KUKA KRL program: MyProgram_082().src

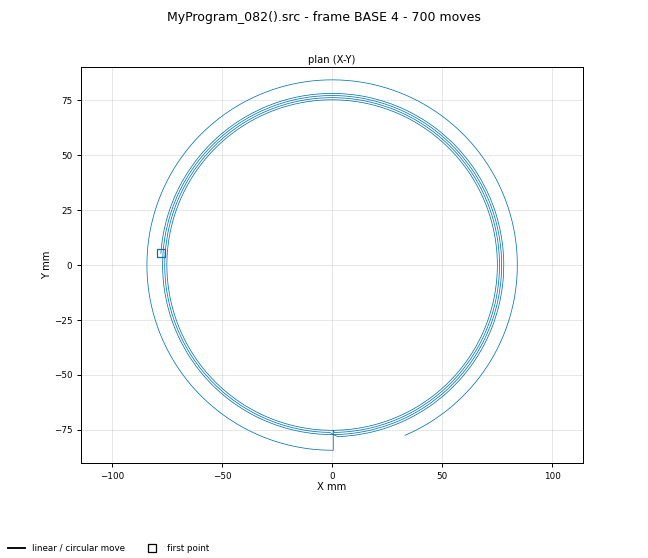
[picture p0: tool path of MyProgram_082().src in frame BASE 4, 700 of 700 moves have a stored position in this frame; points joined in program order, loops and branches not executed]
&ACCESS RVP
&REL 1
&PARAM TEMPLATE = C:\KRC\Roboter\Template\vorgabe
&PARAM EDITMASK = *
DEF MyProgram_082()
; ---- Setting reference (Base) ----
$BASE = BASE_DATA[4]

; --------------------------
; ---- Setting tool (TCP) ----
$TOOL = TOOL_DATA[3]
; --------------------------

$VEL.CP = VEL_APROX_PRINT
Startdeposition()
$VEL.CP = VEL_PRINT
LIN {X -77.8873,Y 5.2841,Z 82,A 170.2718,B 24.9035,C -2.2685,E1 24.8402,E2 274.3605} C_DIS
LIN {X -77.429,Y 9.9551,Z 82,A 166.7128,B 24.9028,C -2.2767,E1 24.8413,E2 277.9213} C_DIS
LIN {X -76.8059,Y 13.9726,Z 82,A 163.8687,B 24.9017,C -2.2896,E1 24.8426,E2 280.7516} C_DIS
LIN {X -76.3731,Y 16.1728,Z 82,A 161.8841,B 24.9019,C -2.2865,E1 24.8437,E2 282.7551} C_DIS
LIN {X -75.4009,Y 20.2256,Z 82,A 158.923,B 24.9009,C -2.2985,E1 24.8457,E2 285.7049} C_DIS
LIN {X -74.3801,Y 23.7078,Z 82,A 156.1268,B 24.9004,C -2.3035,E1 24.848,E2 288.5052} C_DIS
LIN {X -73.114,Y 27.3638,Z 82,A 153.5257,B 24.8992,C -2.318,E1 24.8504,E2 291.0865} C_DIS
LIN {X -71.5308,Y 31.2682,Z 82,A 150.0636,B 24.8992,C -2.3184,E1 24.8542,E2 294.567} C_DIS
LIN {X -69.857,Y 34.848,Z 82,A 147.6109,B 24.8975,C -2.3378,E1 24.8571,E2 296.9865} C_DIS
LIN {X -68.2862,Y 37.834,Z 82,A 144.7243,B 24.8977,C -2.335,E1 24.861,E2 299.8952} C_DIS
LIN {X -65.9152,Y 41.8294,Z 82,A 141.4118,B 24.8966,C -2.3469,E1 24.8657,E2 303.1961} C_DIS
LIN {X -62.1543,Y 47.2375,Z 82,A 136.7737,B 24.8951,C -2.3649,E1 24.8732,E2 307.8141} C_DIS
LIN {X -59.1537,Y 50.9447,Z 82,A 133.0603,B 24.8947,C -2.3686,E1 24.8798,E2 311.5357} C_DIS
LIN {X -56.492,Y 53.8793,Z 82,A 130.0106,B 24.8944,C -2.3723,E1 24.8856,E2 314.5901} C_DIS
LIN {X -53.6602,Y 56.7001,Z 82,A 126.9484,B 24.8941,C -2.376,E1 24.8917,E2 317.6562} C_DIS
LIN {X -50.9442,Y 59.1542,Z 82,A 124.7562,B 24.8924,C -2.3944,E1 24.8963,E2 319.8131} C_DIS
LIN {X -47.0479,Y 62.2967,Z 82,A 120.8026,B 24.8924,C -2.3952,E1 24.9049,E2 323.7796} C_DIS
LIN {X -43.5174,Y 64.8126,Z 82,A 117.5845,B 24.8919,C -2.4006,E1 24.9123,E2 326.9959} C_DIS
LIN {X -40.1757,Y 66.9348,Z 82,A 114.6066,B 24.8915,C -2.4041,E1 24.9194,E2 329.9747} C_DIS
LIN {X -36.2776,Y 69.1252,Z 82,A 111.3707,B 24.8909,C -2.4108,E1 24.9273,E2 333.2038} C_DIS
LIN {X -31.335,Y 71.5017,Z 82,A 107.627,B 24.8897,C -2.4243,E1 24.9367,E2 336.925} C_DIS
LIN {X -29.3343,Y 72.3454,Z 82,A 105.1652,B 24.8915,C -2.404,E1 24.9432,E2 339.4404} C_DIS
LIN {X -26.2143,Y 73.5344,Z 82,A 103.4691,B 24.8895,C -2.4267,E1 24.9475,E2 341.0861} C_DIS
LIN {X -23.2379,Y 74.5276,Z 82,A 100.9819,B 24.8897,C -2.4246,E1 24.9541,E2 343.5828} C_DIS
LIN {X -19.0837,Y 75.6986,Z 82,A 97.8114,B 24.8894,C -2.4277,E1 24.9627,E2 346.7507} C_DIS
LIN {X -15.9587,Y 76.4182,Z 82,A 94.8919,B 24.8906,C -2.4148,E1 24.9707,E2 349.7044} C_DIS
LIN {X -12.813,Y 77.0076,Z 82,A 92.4913,B 24.8906,C -2.4152,E1 24.9773,E2 352.1065} C_DIS
LIN {X -9.4491,Y 77.4932,Z 82,A 90.5626,B 24.889,C -2.4317,E1 24.9826,E2 353.9974} C_DIS
LIN {X -6.2457,Y 77.8161,Z 82,A 88.4719,B 24.8883,C -2.4401,E1 24.9883,E2 356.0689} C_DIS
LIN {X -2.6317,Y 78.0222,Z 82,A 85.4545,B 24.8891,C -2.4313,E1 24.9968,E2 359.1081} C_DIS
LIN {X 1.1853,Y 78.0577,Z 82,A 82.7985,B 24.8887,C -2.4358,E1 25.0042,E2 361.7533} C_DIS
LIN {X 4.2058,Y 77.953,Z 82,A 80.0123,B 24.8901,C -2.4204,E1 25.0121,E2 364.575} C_DIS
LIN {X 9.0381,Y 77.5414,Z 82,A 76.9843,B 24.8888,C -2.4345,E1 25.0204,E2 367.5677} C_DIS
LIN {X 12.3956,Y 77.0774,Z 82,A 74.4767,B 24.8888,C -2.4333,E1 25.0273,E2 370.0759} C_DIS
LIN {X 14.7919,Y 76.6521,Z 82,A 72.0569,B 24.8905,C -2.4151,E1 25.0341,E2 372.5362} C_DIS
LIN {X 18.2659,Y 75.8997,Z 82,A 69.8168,B 24.8897,C -2.4238,E1 25.0401,E2 374.7522} C_DIS
LIN {X 22.1454,Y 74.8594,Z 82,A 67.1483,B 24.8892,C -2.4297,E1 25.0472,E2 377.4025} C_DIS
LIN {X 27.0701,Y 73.2234,Z 82,A 63.363,B 24.8894,C -2.4271,E1 25.0572,E2 381.1863} C_DIS
LIN {X 30.8452,Y 71.7141,Z 82,A 60.3161,B 24.8899,C -2.4223,E1 25.0651,E2 384.2378} C_DIS
LIN {X 33.2005,Y 70.6552,Z 82,A 58.1622,B 24.8908,C -2.4127,E1 25.0706,E2 386.4089} C_DIS
LIN {X 36.1537,Y 69.1905,Z 82,A 55.6058,B 24.8914,C -2.4056,E1 25.0769,E2 388.9749} C_DIS
LIN {X 40.9292,Y 66.4769,Z 82,A 51.804,B 24.8914,C -2.4064,E1 25.086,E2 392.7631} C_DIS
LIN {X 43.8416,Y 64.5931,Z 82,A 49.597,B 24.8908,C -2.4122,E1 25.0911,E2 394.9491} C_DIS
LIN {X 46.4973,Y 62.7102,Z 82,A 47.0872,B 24.8915,C -2.4045,E1 25.0968,E2 397.4681} C_DIS
LIN {X 49.1805,Y 60.627,Z 82,A 44.682,B 24.8917,C -2.4026,E1 25.1021,E2 399.8689} C_DIS
LIN {X 53.8052,Y 56.5645,Z 82,A 40.1147,B 24.8926,C -2.3922,E1 25.1116,E2 404.4426} C_DIS
LIN {X 55.3996,Y 55.0025,Z 82,A 37.5288,B 24.8954,C -2.3608,E1 25.1168,E2 407.0916} C_DIS
LIN {X 58.5315,Y 51.6583,Z 82,A 35.1537,B 24.8935,C -2.3825,E1 25.1211,E2 409.405} C_DIS
LIN {X 62.0522,Y 47.3708,Z 82,A 31.4627,B 24.8933,C -2.3843,E1 25.1275,E2 413.0744} C_DIS
LIN {X 64.4349,Y 44.0753,Z 82,A 28.1614,B 24.8948,C -2.3674,E1 25.1329,E2 416.3998} C_DIS
LIN {X 66.1554,Y 41.4466,Z 82,A 25.946,B 24.8951,C -2.3642,E1 25.1362,E2 418.6115} C_DIS
LIN {X 67.7327,Y 38.8154,Z 82,A 23.6134,B 24.8959,C -2.3558,E1 25.1395,E2 420.952} C_DIS
LIN {X 70.3142,Y 33.9156,Z 82,A 20.0711,B 24.8954,C -2.3606,E1 25.1441,E2 424.4642} C_DIS
LIN {X 71.9062,Y 30.395,Z 82,A 16.8555,B 24.8972,C -2.341,E1 25.1478,E2 427.7087} C_DIS
LIN {X 72.9013,Y 27.9255,Z 82,A 14.8235,B 24.8979,C -2.3329,E1 25.1498,E2 429.7484} C_DIS
LIN {X 73.9869,Y 24.9056,Z 82,A 12.4921,B 24.8984,C -2.3267,E1 25.152,E2 432.0813} C_DIS
LIN {X 74.87,Y 22.1096,Z 82,A 9.9478,B 24.9,C -2.3083,E1 25.154,E2 434.6547} C_DIS
LIN {X 76.297,Y 16.5264,Z 82,A 5.6468,B 24.9013,C -2.2932,E1 25.1568,E2 438.9663} C_DIS
LIN {X 77.1156,Y 12.1461,Z 82,A 2.8117,B 24.9011,C -2.2965,E1 25.1581,E2 441.7772} C_DIS
LIN {X 77.5907,Y 8.6165,Z 82,A 0.0655,B 24.9021,C -2.2842,E1 25.1591,E2 444.5362} C_DIS
LIN {X 77.9848,Y 3.5743,Z 82,A -3.4052,B 24.9025,C -2.2799,E1 25.1597,E2 447.9965} C_DIS
LIN {X 78.0657,Y 0.3664,Z 82,A -5.5988,B 24.9027,C -2.2774,E1 25.1597,E2 450.1828} C_DIS
LIN {X 77.93,Y -4.6221,Z 82,A -9.3508,B 24.9039,C -2.2629,E1 25.1594,E2 453.9467} C_DIS
LIN {X 77.7316,Y -7.2215,Z 82,A -12.3122,B 24.9072,C -2.2246,E1 25.1586,E2 456.981} C_DIS
LIN {X 77.1522,Y -11.9113,Z 82,A -14.1609,B 24.9039,C -2.2635,E1 25.1579,E2 458.727} C_DIS
LIN {X 76.2149,Y -16.9028,Z 82,A -18.366,B 24.9061,C -2.2368,E1 25.1557,E2 462.9706} C_DIS
LIN {X 75.4606,Y -20.0044,Z 82,A -21.1675,B 24.9079,C -2.2153,E1 25.1537,E2 465.8068} C_DIS
LIN {X 73.6511,Y -25.8816,Z 82,A -25.0046,B 24.9074,C -2.2222,E1 25.1505,E2 469.6058} C_DIS
LIN {X 72.5926,Y -28.7174,Z 82,A -27.7071,B 24.9092,C -2.2005,E1 25.1477,E2 472.3443} C_DIS
LIN {X 70.4919,Y -33.5459,Z 82,A -31.2442,B 24.9092,C -2.199,E1 25.1437,E2 475.8658} C_DIS
LIN {X 68.5885,Y -37.2823,Z 82,A -34.6146,B 24.9108,C -2.1811,E1 25.1393,E2 479.2608} C_DIS
LIN {X 66.523,Y -40.8554,Z 82,A -37.3547,B 24.9108,C -2.1813,E1 25.1354,E2 481.9865} C_DIS
LIN {X 64.3814,Y -44.1542,Z 82,A -40.9192,B 24.9131,C -2.1526,E1 25.1297,E2 485.6009} C_DIS
LIN {X 62.2055,Y -47.1689,Z 82,A -43.079,B 24.9123,C -2.1626,E1 25.1262,E2 487.7269} C_DIS
LIN {X 60.5533,Y -49.2714,Z 82,A -45.6835,B 24.9143,C -2.138,E1 25.1215,E2 490.3773} C_DIS
LIN {X 57.8989,Y -52.3663,Z 82,A -47.3704,B 24.9117,C -2.17,E1 25.1185,E2 491.9812} C_DIS
LIN {X 54.1289,Y -56.2532,Z 82,A -51.2413,B 24.9122,C -2.1634,E1 25.111,E2 495.8511} C_DIS
LIN {X 51.7209,Y -58.4767,Z 82,A -54.1763,B 24.914,C -2.1417,E1 25.1049,E2 498.8254} C_DIS
LIN {X 50.0399,Y -59.9199,Z 82,A -56.6865,B 24.9164,C -2.1117,E1 25.0993,E2 501.3969} C_DIS
LIN {X 46.7247,Y -62.5396,Z 82,A -58.6933,B 24.9143,C -2.1378,E1 25.095,E2 503.3348} C_DIS
LIN {X 44.4197,Y -64.1966,Z 82,A -61.5923,B 24.9166,C -2.1093,E1 25.0883,E2 506.2912} C_DIS
LIN {X 41.5013,Y -66.1212,Z 82,A -63.0694,B 24.9144,C -2.1367,E1 25.085,E2 507.6985} C_DIS
LIN {X 39.5834,Y -67.2869,Z 82,A -65.7493,B 24.917,C -2.1031,E1 25.0783,E2 510.4498} C_DIS
LIN {X 36.6318,Y -68.9387,Z 82,A -67.7374,B 24.9162,C -2.1134,E1 25.0735,E2 512.4079} C_DIS
LIN {X 33.2308,Y -70.6411,Z 82,A -70.4044,B 24.9162,C -2.1126,E1 25.0668,E2 515.0698} C_DIS
LIN {X 30.2504,Y -71.9671,Z 82,A -72.9473,B 24.9169,C -2.1047,E1 25.0603,E2 517.6252} C_DIS
LIN {X 26.1878,Y -73.5436,Z 82,A -76.2474,B 24.9175,C -2.0975,E1 25.0516,E2 520.9354} C_DIS
LIN {X 23.3601,Y -74.4897,Z 82,A -78.4432,B 24.9177,C -2.0947,E1 25.0458,E2 523.1338} C_DIS
LIN {X 19.1921,Y -75.6708,Z 82,A -81.3872,B 24.9174,C -2.0981,E1 25.0379,E2 526.0649} C_DIS
LIN {X 15.9256,Y -76.425,Z 82,A -83.7655,B 24.9174,C -2.0983,E1 25.0314,E2 528.4398} C_DIS
LIN {X 9.9884,Y -77.4247,Z 82,A -87.7279,B 24.9167,C -2.1081,E1 25.0206,E2 532.3749} C_DIS
LIN {X 5.5408,Y -77.8699,Z 82,A -91.4789,B 24.9179,C -2.0929,E1 25.01,E2 536.1596} C_DIS
LIN {X 2.6008,Y -78.0232,Z 82,A -94.2473,B 24.9192,C -2.0752,E1 25.0022,E2 538.9694} C_DIS
LIN {X 2.6008,Y -78.0232,Z 82,A -94.2473,B 24.9192,C -2.0752,E1 25.0022,E2 538.9694} C_DIS
Enddeposition()
LIN {X 0.5081,Y -77.0915,Z 82,A -94.1358,B 24.9143,C -2.1379,E1 25.0029,E2 538.7091} C_DIS
Startdeposition()
$VEL.CP = VEL_PRINT
LIN {X 3.9501,Y -76.9968,Z 82,A -91.5866,B 24.9143,C -2.1385,E1 25.01,E2 536.1593} C_DIS
LIN {X 6.6748,Y -76.8091,Z 82,A -88.9999,B 24.9129,C -2.1554,E1 25.0173,E2 533.5338} C_DIS
LIN {X 10.5371,Y -76.3746,Z 82,A -86.2088,B 24.9129,C -2.1544,E1 25.0251,E2 530.7472} C_DIS
LIN {X 14.7289,Y -75.6776,Z 82,A -83.4663,B 24.9137,C -2.1449,E1 25.0325,E2 528.0303} C_DIS
LIN {X 17.832,Y -75.0082,Z 82,A -81.0789,B 24.9135,C -2.1479,E1 25.039,E2 525.6391} C_DIS
LIN {X 23.2313,Y -73.5153,Z 82,A -77.1971,B 24.9138,C -2.1443,E1 25.0494,E2 521.7725} C_DIS
LIN {X 28.0703,Y -71.8059,Z 82,A -73.1834,B 24.9129,C -2.1551,E1 25.06,E2 517.7415} C_DIS
LIN {X 30.9867,Y -70.5966,Z 82,A -70.8936,B 24.9128,C -2.1568,E1 25.0659,E2 515.4531} C_DIS
LIN {X 33.8173,Y -69.2864,Z 82,A -68.4579,B 24.9122,C -2.1639,E1 25.072,E2 513.0068} C_DIS
LIN {X 36.6293,Y -67.8405,Z 82,A -66.4322,B 24.9126,C -2.1583,E1 25.077,E2 511.0001} C_DIS
LIN {X 39.8423,Y -66.005,Z 82,A -63.7443,B 24.9124,C -2.1614,E1 25.0835,E2 508.313} C_DIS
LIN {X 42.2071,Y -64.5186,Z 82,A -61.3442,B 24.9113,C -2.175,E1 25.0892,E2 505.8885} C_DIS
LIN {X 44.9897,Y -62.61,Z 82,A -58.5122,B 24.91,C -2.1899,E1 25.0957,E2 503.0311} C_DIS
LIN {X 49.3722,Y -59.215,Z 82,A -54.9467,B 24.9107,C -2.182,E1 25.1034,E2 499.4976} C_DIS
LIN {X 51.4404,Y -57.4274,Z 82,A -52.997,B 24.9105,C -2.1841,E1 25.1075,E2 497.5506} C_DIS
LIN {X 53.2707,Y -55.7347,Z 82,A -50.8786,B 24.9095,C -2.1965,E1 25.1119,E2 495.4115} C_DIS
LIN {X 57.0794,Y -51.8277,Z 82,A -47.2458,B 24.9097,C -2.1936,E1 25.1189,E2 491.8013} C_DIS
LIN {X 60.3106,Y -48.0284,Z 82,A -42.4331,B 24.9061,C -2.2372,E1 25.1276,E2 486.9077} C_DIS
LIN {X 62.5808,Y -45.0302,Z 82,A -40.2831,B 24.9071,C -2.2248,E1 25.131,E2 484.7974} C_DIS
LIN {X 64.3492,Y -42.464,Z 82,A -37.5283,B 24.9055,C -2.2448,E1 25.1353,E2 482.009} C_DIS
LIN {X 66.0971,Y -39.6896,Z 82,A -35.7395,B 24.9066,C -2.2316,E1 25.1379,E2 480.2605} C_DIS
LIN {X 68.7522,Y -34.8884,Z 82,A -31.5814,B 24.9054,C -2.246,E1 25.1434,E2 476.0903} C_DIS
LIN {X 70.1743,Y -31.9321,Z 82,A -29.217,B 24.9049,C -2.2509,E1 25.1462,E2 473.7269} C_DIS
LIN {X 72.3496,Y -26.6385,Z 82,A -25.1385,B 24.9043,C -2.2584,E1 25.1504,E2 469.6533} C_DIS
LIN {X 73.4824,Y -23.335,Z 82,A -22.2849,B 24.9029,C -2.2744,E1 25.1529,E2 466.778} C_DIS
LIN {X 74.4554,Y -20.0105,Z 82,A -19.8348,B 24.9026,C -2.2786,E1 25.1548,E2 464.332} C_DIS
LIN {X 75.2068,Y -16.9735,Z 82,A -17.55,B 24.9021,C -2.2847,E1 25.1562,E2 462.0463} C_DIS
LIN {X 76.0528,Y -12.649,Z 82,A -14.4847,B 24.9017,C -2.2886,E1 25.1578,E2 458.9898} C_DIS
LIN {X 76.6432,Y -8.3636,Z 82,A -11.2642,B 24.9008,C -2.299,E1 25.159,E2 455.7637} C_DIS
LIN {X 76.8675,Y -5.953,Z 82,A -9.3343,B 24.9,C -2.3088,E1 25.1594,E2 453.8221} C_DIS
LIN {X 77.0423,Y -2.9386,Z 82,A -6.7313,B 24.8984,C -2.3271,E1 25.1597,E2 451.1911} C_DIS
LIN {X 77.0463,Y 2.8462,Z 82,A -3.0401,B 24.8989,C -2.3218,E1 25.1597,E2 447.5344} C_DIS
LIN {X 76.9112,Y 5.3576,Z 82,A -0.7479,B 24.8972,C -2.3409,E1 25.1592,E2 445.2108} C_DIS
LIN {X 76.5442,Y 9.2231,Z 82,A 2.5236,B 24.8953,C -2.362,E1 25.1582,E2 441.9087} C_DIS
LIN {X 76.0708,Y 12.541,Z 82,A 4.0458,B 24.8973,C -2.3397,E1 25.1576,E2 440.4483} C_DIS
LIN {X 75.6164,Y 15.0462,Z 82,A 7.107,B 24.8935,C -2.3818,E1 25.1559,E2 437.3054} C_DIS
LIN {X 74.7352,Y 18.9403,Z 82,A 8.8697,B 24.8961,C -2.3535,E1 25.1548,E2 435.6199} C_DIS
LIN {X 74.0877,Y 21.3339,Z 82,A 10.8114,B 24.8953,C -2.3621,E1 25.1533,E2 433.6691} C_DIS
LIN {X 73.3737,Y 23.6709,Z 82,A 12.8236,B 24.8943,C -2.3735,E1 25.1516,E2 431.6412} C_DIS
LIN {X 72.4155,Y 26.4578,Z 82,A 15.0029,B 24.8937,C -2.3796,E1 25.1495,E2 429.4598} C_DIS
LIN {X 71.3013,Y 29.3295,Z 82,A 17.6471,B 24.8922,C -2.3971,E1 25.1468,E2 426.7888} C_DIS
LIN {X 69.697,Y 32.9631,Z 82,A 20.2218,B 24.8925,C -2.3938,E1 25.1438,E2 424.236} C_DIS
LIN {X 67.8475,Y 36.6165,Z 82,A 22.9827,B 24.8925,C -2.3935,E1 25.1403,E2 421.4903} C_DIS
LIN {X 66.5797,Y 38.8758,Z 82,A 25.2155,B 24.8912,C -2.408,E1 25.1371,E2 419.235} C_DIS
LIN {X 64.7601,Y 41.8353,Z 82,A 27.5063,B 24.8914,C -2.4058,E1 25.1338,E2 416.9608} C_DIS
LIN {X 62.4871,Y 45.1598,Z 82,A 31.2112,B 24.8887,C -2.4349,E1 25.1277,E2 413.2053} C_DIS
LIN {X 59.1541,Y 49.4455,Z 82,A 34.5329,B 24.8898,C -2.4228,E1 25.122,E2 409.9276} C_DIS
LIN {X 57.415,Y 51.4542,Z 82,A 37.2241,B 24.8875,C -2.4488,E1 25.1169,E2 407.1869} C_DIS
LIN {X 53.7515,Y 55.2712,Z 82,A 40.6308,B 24.8881,C -2.4413,E1 25.1103,E2 403.8124} C_DIS
LIN {X 50.1748,Y 58.5368,Z 82,A 43.9057,B 24.8884,C -2.4388,E1 25.1035,E2 400.5565} C_DIS
LIN {X 48.2335,Y 60.1473,Z 82,A 46.0869,B 24.8872,C -2.4513,E1 25.0988,E2 398.354} C_DIS
LIN {X 45.8494,Y 61.9838,Z 82,A 48.3638,B 24.8867,C -2.4564,E1 25.0937,E2 396.0732} C_DIS
LIN {X 43.0679,Y 63.9469,Z 82,A 50.4983,B 24.8874,C -2.449,E1 25.0888,E2 393.9635} C_DIS
LIN {X 41.2641,Y 65.1268,Z 82,A 53.0326,B 24.8847,C -2.4788,E1 25.0827,E2 391.3669} C_DIS
LIN {X 38.4025,Y 66.8526,Z 82,A 55.4751,B 24.8845,C -2.4811,E1 25.0768,E2 388.9263} C_DIS
LIN {X 35.4552,Y 68.4625,Z 82,A 57.1028,B 24.8865,C -2.4591,E1 25.0729,E2 387.3552} C_DIS
LIN {X 33.035,Y 69.6625,Z 82,A 59.1236,B 24.8862,C -2.462,E1 25.0679,E2 385.3331} C_DIS
LIN {X 31.0756,Y 70.5578,Z 82,A 61.266,B 24.8846,C -2.4793,E1 25.0623,E2 383.1549} C_DIS
LIN {X 27.7636,Y 71.9264,Z 82,A 63.8133,B 24.8846,C -2.4786,E1 25.0557,E2 380.615} C_DIS
LIN {X 24.1282,Y 73.2258,Z 82,A 66.5464,B 24.8848,C -2.4771,E1 25.0485,E2 377.8906} C_DIS
LIN {X 19.882,Y 74.4901,Z 82,A 69.9019,B 24.8844,C -2.4812,E1 25.0395,E2 374.5312} C_DIS
LIN {X 15.6334,Y 75.4959,Z 82,A 72.5546,B 24.8858,C -2.4663,E1 25.0324,E2 371.9175} C_DIS
LIN {X 13.5841,Y 75.8913,Z 82,A 74.5578,B 24.8846,C -2.4795,E1 25.0268,E2 369.8852} C_DIS
LIN {X 10.6196,Y 76.3629,Z 82,A 76.7717,B 24.8846,C -2.4795,E1 25.0207,E2 367.6731} C_DIS
LIN {X 6.6725,Y 76.8088,Z 82,A 79.939,B 24.884,C -2.4859,E1 25.0118,E2 364.4928} C_DIS
LIN {X 3.8251,Y 77.0037,Z 82,A 81.9048,B 24.8844,C -2.4816,E1 25.0064,E2 362.5381} C_DIS
LIN {X 0.5366,Y 77.0956,Z 82,A 84.2089,B 24.8848,C -2.4774,E1 25,E2 360.2442} C_DIS
LIN {X -3.2844,Y 77.0275,Z 82,A 87.365,B 24.8841,C -2.4852,E1 24.9911,E2 357.0691} C_DIS
LIN {X -7.1127,Y 76.7687,Z 82,A 90.01,B 24.8847,C -2.4783,E1 24.9838,E2 354.4393} C_DIS
LIN {X -10.3824,Y 76.3966,Z 82,A 92.8584,B 24.8838,C -2.4877,E1 24.9758,E2 351.5666} C_DIS
LIN {X -15.1482,Y 75.5955,Z 82,A 95.7569,B 24.8858,C -2.4665,E1 24.968,E2 348.7156} C_DIS
LIN {X -17.6309,Y 75.055,Z 82,A 98.0189,B 24.8851,C -2.4747,E1 24.9618,E2 346.4311} C_DIS
LIN {X -20.9974,Y 74.183,Z 82,A 101.3824,B 24.8834,C -2.4928,E1 24.9526,E2 343.0193} C_DIS
LIN {X -24.8215,Y 72.9928,Z 82,A 103.2877,B 24.8863,C -2.4609,E1 24.9478,E2 341.1863} C_DIS
LIN {X -27.3843,Y 72.0702,Z 82,A 106.0937,B 24.8847,C -2.4788,E1 24.9403,E2 338.3318} C_DIS
LIN {X -32.2108,Y 70.0461,Z 82,A 109.7731,B 24.8857,C -2.4676,E1 24.9309,E2 334.6704} C_DIS
LIN {X -35.2561,Y 68.5643,Z 82,A 111.9235,B 24.887,C -2.4541,E1 24.9256,E2 332.5465} C_DIS
LIN {X -38.1112,Y 67.02,Z 82,A 114.8426,B 24.8861,C -2.463,E1 24.9185,E2 329.5977} C_DIS
LIN {X -41.7966,Y 64.7849,Z 82,A 117.5941,B 24.8878,C -2.4454,E1 24.912,E2 326.8793} C_DIS
LIN {X -44.3849,Y 63.0413,Z 82,A 120.0434,B 24.8878,C -2.4442,E1 24.9064,E2 324.4248} C_DIS
LIN {X -47.1418,Y 61.0055,Z 82,A 123.3863,B 24.8865,C -2.4592,E1 24.8989,E2 321.0337} C_DIS
LIN {X -50.3449,Y 58.3919,Z 82,A 125.3766,B 24.8896,C -2.4249,E1 24.8948,E2 319.1176} C_DIS
LIN {X -54.3022,Y 54.7295,Z 82,A 129.1584,B 24.891,C -2.41,E1 24.8871,E2 315.3559} C_DIS
LIN {X -57.8188,Y 51.0014,Z 82,A 133.4368,B 24.8908,C -2.4122,E1 24.8789,E2 311.0535} C_DIS
LIN {X -60.9616,Y 47.1988,Z 82,A 137.1674,B 24.8915,C -2.4043,E1 24.8724,E2 307.3244} C_DIS
LIN {X -63.7522,Y 43.3554,Z 82,A 140.5843,B 24.8926,C -2.392,E1 24.8669,E2 303.9202} C_DIS
LIN {X -65.29,Y 41.0033,Z 82,A 142.7697,B 24.8929,C -2.3885,E1 24.8636,E2 301.732} C_DIS
LIN {X -67.6657,Y 36.9516,Z 82,A 146.3026,B 24.8937,C -2.3796,E1 24.8587,E2 298.2021} C_DIS
LIN {X -69.1522,Y 34.0884,Z 82,A 148.7057,B 24.8944,C -2.3727,E1 24.8556,E2 295.8024} C_DIS
LIN {X -70.5534,Y 31.0858,Z 82,A 152.1596,B 24.8928,C -2.3899,E1 24.8517,E2 292.2886} C_DIS
LIN {X -72.1749,Y 27.108,Z 82,A 154.2774,B 24.8961,C -2.3537,E1 24.8496,E2 290.2454} C_DIS
LIN {X -73.3992,Y 23.5922,Z 82,A 157.5107,B 24.8958,C -2.3565,E1 24.8467,E2 286.9868} C_DIS
LIN {X -74.3415,Y 20.4323,Z 82,A 160.0168,B 24.8964,C -2.3503,E1 24.8448,E2 284.4811} C_DIS
LIN {X -75.5252,Y 15.4907,Z 82,A 163.3487,B 24.8984,C -2.3275,E1 24.8428,E2 281.1839} C_DIS
LIN {X -76.0455,Y 12.6924,Z 82,A 165.7516,B 24.8984,C -2.3278,E1 24.8416,E2 278.7661} C_DIS
LIN {X -76.5929,Y 8.8073,Z 82,A 168.7267,B 24.899,C -2.32,E1 24.8406,E2 275.7919} C_DIS
LIN {X -76.9455,Y 4.851,Z 82,A 171.6104,B 24.9,C -2.3089,E1 24.84,E2 272.9173} C_DIS
LIN {X -77.0936,Y 0.8846,Z 82,A 174.558,B 24.9008,C -2.2995,E1 24.8398,E2 269.9746} C_DIS
LIN {X -77.0556,Y -2.5454,Z 82,A 176.9796,B 24.9018,C -2.2883,E1 24.8399,E2 267.5651} C_DIS
LIN {X -76.8971,Y -5.5662,Z 82,A 179.4264,B 24.902,C -2.286,E1 24.8404,E2 265.1089} C_DIS
LIN {X -76.5566,Y -9.1173,Z 82,A -178.0985,B 24.903,C -2.2734,E1 24.8411,E2 262.6492} C_DIS
LIN {X -76.1375,Y -12.1339,Z 82,A -175.6368,B 24.9032,C -2.2712,E1 24.8421,E2 260.1781} C_DIS
LIN {X -75.4419,Y -15.8904,Z 82,A -172.8899,B 24.9042,C -2.2602,E1 24.8436,E2 257.4411} C_DIS
LIN {X -74.9446,Y -18.0929,Z 82,A -170.27,B 24.9026,C -2.2785,E1 24.8454,E2 254.7624} C_DIS
LIN {X -73.8516,Y -22.1361,Z 82,A -168.2018,B 24.9056,C -2.2432,E1 24.8469,E2 252.7664} C_DIS
LIN {X -73.0767,Y -24.5727,Z 82,A -166.0197,B 24.9055,C -2.2446,E1 24.8488,E2 250.5686} C_DIS
LIN {X -71.918,Y -27.7851,Z 82,A -162.5058,B 24.904,C -2.2616,E1 24.8524,E2 246.9941} C_DIS
LIN {X -70.1116,Y -32.0713,Z 82,A -160.0262,B 24.9069,C -2.2273,E1 24.8552,E2 244.5829} C_DIS
LIN {X -68.8561,Y -34.6851,Z 82,A -157.8851,B 24.9075,C -2.2211,E1 24.8578,E2 242.4452} C_DIS
LIN {X -65.8797,Y -40.0484,Z 82,A -153.5584,B 24.909,C -2.2031,E1 24.8638,E2 238.1386} C_DIS
LIN {X -64.4775,Y -42.2695,Z 82,A -150.3245,B 24.9067,C -2.2307,E1 24.8689,E2 234.8228} C_DIS
LIN {X -61.8304,Y -46.0556,Z 82,A -147.9294,B 24.9096,C -2.1958,E1 24.8727,E2 232.4994} C_DIS
LIN {X -59.8455,Y -48.606,Z 82,A -145.467,B 24.9099,C -2.1917,E1 24.877,E2 230.0352} C_DIS
LIN {X -57.9953,Y -50.7993,Z 82,A -142.8851,B 24.9093,C -2.1984,E1 24.8817,E2 227.4256} C_DIS
LIN {X -54.9121,Y -54.1173,Z 82,A -139.976,B 24.9109,C -2.1794,E1 24.8873,E2 224.5492} C_DIS
LIN {X -52.806,Y -56.1742,Z 82,A -137.2537,B 24.9101,C -2.1888,E1 24.8929,E2 221.7933} C_DIS
LIN {X -49.689,Y -58.9507,Z 82,A -134.6452,B 24.9117,C -2.17,E1 24.8983,E2 219.2194} C_DIS
LIN {X -47.1515,Y -60.9981,Z 82,A -131.6207,B 24.9107,C -2.1814,E1 24.9051,E2 216.1565} C_DIS
LIN {X -44.395,Y -63.0343,Z 82,A -129.1858,B 24.9113,C -2.1742,E1 24.9106,E2 213.7304} C_DIS
LIN {X -40.1524,Y -65.8165,Z 82,A -125.6154,B 24.9122,C -2.1633,E1 24.919,E2 210.1748} C_DIS
LIN {X -37.2718,Y -67.4905,Z 82,A -123.3806,B 24.913,C -2.1535,E1 24.9244,E2 207.9568} C_DIS
LIN {X -34.4211,Y -68.9873,Z 82,A -120.3806,B 24.9119,C -2.1668,E1 24.932,E2 204.9171} C_DIS
LIN {X -31.3077,Y -70.4555,Z 82,A -118.7273,B 24.9141,C -2.1396,E1 24.936,E2 203.3244} C_DIS
LIN {X -29.2523,Y -71.3327,Z 82,A -116.6037,B 24.9133,C -2.1504,E1 24.9416,E2 201.1703} C_DIS
LIN {X -25.4811,Y -72.7649,Z 82,A -113.5102,B 24.9133,C -2.1504,E1 24.9497,E2 198.0706} C_DIS
LIN {X -20.957,Y -74.1945,Z 82,A -109.8457,B 24.9132,C -2.1517,E1 24.9596,E2 194.3968} C_DIS
LIN {X -16.8908,Y -75.2258,Z 82,A -107.1236,B 24.9142,C -2.1392,E1 24.9669,E2 191.7008} C_DIS
LIN {X -13.867,Y -75.8404,Z 82,A -104.8342,B 24.9142,C -2.1383,E1 24.9732,E2 189.4111} C_DIS
LIN {X -9.6224,Y -76.4951,Z 82,A -101.3076,B 24.9136,C -2.1469,E1 24.983,E2 185.8612} C_DIS
LIN {X -5.6504,Y -76.8914,Z 82,A -98.6106,B 24.9142,C -2.1392,E1 24.9904,E2 183.1812} C_DIS
LIN {X -2.3423,Y -77.0619,Z 82,A -95.9455,B 24.9137,C -2.1452,E1 24.9979,E2 180.5014} C_DIS
LIN {X 0.5081,Y -77.0915,Z 82,A -94.1339,B 24.9143,C -2.1371,E1 25.0029,E2 178.7091} C_DIS
Enddeposition()
LIN {X 0.5081,Y -77.0915,Z 82,A -94.1339,B 24.9143,C -2.1371,E1 25.0029,E2 178.7091} C_DIS
Startdeposition()
$VEL.CP = VEL_PRINT
LIN {X -1.1038,Y -76.1212,Z 82,A -96.4432,B 24.9155,C -2.1232,E1 24.9964,E2 181.0513} C_DIS
LIN {X -4.2438,Y -76.0102,Z 82,A -98.8012,B 24.9155,C -2.1232,E1 24.9898,E2 183.4099} C_DIS
LIN {X -7.3852,Y -75.7705,Z 82,A -101.1105,B 24.9153,C -2.125,E1 24.9834,E2 185.7161} C_DIS
LIN {X -10.3028,Y -75.4293,Z 82,A -103.3603,B 24.9153,C -2.1243,E1 24.9771,E2 187.9691} C_DIS
LIN {X -12.9873,Y -75.0139,Z 82,A -105.4319,B 24.9153,C -2.1242,E1 24.9714,E2 190.043} C_DIS
LIN {X -15.9653,Y -74.4361,Z 82,A -107.7339,B 24.9153,C -2.1246,E1 24.9651,E2 192.3466} C_DIS
LIN {X -19.1563,Y -73.6793,Z 82,A -110.1969,B 24.9153,C -2.1261,E1 24.9584,E2 194.8095} C_DIS
LIN {X -22.2641,Y -72.8008,Z 82,A -113.4199,B 24.9167,C -2.1071,E1 24.9497,E2 198.083} C_DIS
LIN {X -25.8483,Y -71.6065,Z 82,A -115.7987,B 24.9156,C -2.1215,E1 24.9435,E2 200.4323} C_DIS
LIN {X -29.6391,Y -70.122,Z 82,A -118.6058,B 24.9148,C -2.1312,E1 24.9363,E2 203.2225} C_DIS
LIN {X -33.6955,Y -68.2656,Z 82,A -121.8468,B 24.9143,C -2.1381,E1 24.9281,E2 206.4554} C_DIS
LIN {X -36.3543,Y -66.8875,Z 82,A -123.9823,B 24.9138,C -2.144,E1 24.9229,E2 208.5827} C_DIS
LIN {X -40.4863,Y -64.4706,Z 82,A -127.7979,B 24.9138,C -2.1437,E1 24.9137,E2 212.4106} C_DIS
LIN {X -43.0643,Y -62.7791,Z 82,A -130.1727,B 24.9136,C -2.146,E1 24.9082,E2 214.7878} C_DIS
LIN {X -45.0341,Y -61.3799,Z 82,A -132.1209,B 24.9136,C -2.1459,E1 24.9038,E2 216.7433} C_DIS
LIN {X -47.941,Y -59.1373,Z 82,A -134.7189,B 24.9129,C -2.155,E1 24.8981,E2 219.3292} C_DIS
LIN {X -49.7768,Y -57.602,Z 82,A -137.2905,B 24.9142,C -2.1393,E1 24.8926,E2 221.9482} C_DIS
LIN {X -52.5194,Y -55.1131,Z 82,A -139.4131,B 24.9124,C -2.1613,E1 24.8883,E2 224.0272} C_DIS
LIN {X -54.8674,Y -52.7743,Z 82,A -141.4919,B 24.9111,C -2.1768,E1 24.8843,E2 226.0777} C_DIS
LIN {X -57.5803,Y -49.8016,Z 82,A -144.5728,B 24.9107,C -2.1822,E1 24.8785,E2 229.1595} C_DIS
LIN {X -59.9753,Y -46.8901,Z 82,A -147.616,B 24.9106,C -2.1838,E1 24.8732,E2 232.2131} C_DIS
LIN {X -62.2674,Y -43.8008,Z 82,A -150.7106,B 24.9104,C -2.186,E1 24.8681,E2 235.3175} C_DIS
LIN {X -64.0528,Y -41.1436,Z 82,A -152.946,B 24.9095,C -2.1963,E1 24.8646,E2 237.5395} C_DIS
LIN {X -65.5236,Y -38.7585,Z 82,A -155.0489,B 24.9091,C -2.2019,E1 24.8616,E2 239.6397} C_DIS
LIN {X -67.2626,Y -35.6559,Z 82,A -157.81,B 24.9086,C -2.2071,E1 24.8579,E2 242.4031} C_DIS
LIN {X -68.4668,Y -33.2864,Z 82,A -159.9208,B 24.9084,C -2.2099,E1 24.8553,E2 244.5184} C_DIS
LIN {X -70.1668,Y -29.5328,Z 82,A -163.0182,B 24.9077,C -2.2188,E1 24.8518,E2 247.6117} C_DIS
LIN {X -71.3749,Y -26.4832,Z 82,A -165.3887,B 24.9069,C -2.2282,E1 24.8494,E2 249.973} C_DIS
LIN {X -72.6497,Y -22.7515,Z 82,A -168.4579,B 24.9063,C -2.2346,E1 24.8467,E2 253.0445} C_DIS
LIN {X -73.5196,Y -19.7596,Z 82,A -171.2302,B 24.9066,C -2.2316,E1 24.8446,E2 255.8402} C_DIS
LIN {X -74.2607,Y -16.7645,Z 82,A -173.5501,B 24.906,C -2.2387,E1 24.8432,E2 258.1567} C_DIS
LIN {X -75.0464,Y -12.7931,Z 82,A -176.232,B 24.9045,C -2.2566,E1 24.8418,E2 260.8116} C_DIS
LIN {X -75.5002,Y -9.7612,Z 82,A -178.5431,B 24.9039,C -2.2638,E1 24.8409,E2 263.1195} C_DIS
LIN {X -75.8475,Y -6.5508,Z 82,A 178.8854,B 24.9035,C -2.2681,E1 24.8402,E2 265.6962} C_DIS
LIN {X -76.0581,Y -3.2761,Z 82,A 176.6134,B 24.9024,C -2.2805,E1 24.8399,E2 267.952} C_DIS
LIN {X -76.1275,Y -0.457,Z 82,A 174.3777,B 24.9021,C -2.2846,E1 24.8398,E2 270.1914} C_DIS
LIN {X -76.093,Y 2.3286,Z 82,A 172.2402,B 24.9016,C -2.2903,E1 24.8399,E2 272.3282} C_DIS
LIN {X -75.9285,Y 5.5293,Z 82,A 170.0202,B 24.9005,C -2.3025,E1 24.8403,E2 274.5324} C_DIS
LIN {X -75.7442,Y 7.6423,Z 82,A 167.6372,B 24.9017,C -2.2892,E1 24.841,E2 276.9614} C_DIS
LIN {X -74.8601,Y 13.8446,Z 82,A 163.6669,B 24.8989,C -2.3216,E1 24.8426,E2 280.8781} C_DIS
LIN {X -74.1373,Y 17.299,Z 82,A 160.2344,B 24.8997,C -2.3118,E1 24.8447,E2 284.3541} C_DIS
LIN {X -73.2757,Y 20.6457,Z 82,A 157.559,B 24.8992,C -2.3182,E1 24.8468,E2 287.0299} C_DIS
LIN {X -72.3265,Y 23.7605,Z 82,A 155.6664,B 24.8974,C -2.3387,E1 24.8483,E2 288.8842} C_DIS
LIN {X -71.2614,Y 26.7844,Z 82,A 153.2758,B 24.8967,C -2.3466,E1 24.8506,E2 291.2694} C_DIS
LIN {X -70.4557,Y 28.837,Z 82,A 151.3629,B 24.8967,C -2.3457,E1 24.8526,E2 293.1953} C_DIS
LIN {X -68.9697,Y 32.2298,Z 82,A 148.7727,B 24.8956,C -2.3586,E1 24.8556,E2 295.7687} C_DIS
LIN {X -67.6279,Y 34.9594,Z 82,A 146.5671,B 24.8948,C -2.3673,E1 24.8584,E2 297.9654} C_DIS
LIN {X -66.2025,Y 37.5891,Z 82,A 144.1623,B 24.8946,C -2.3701,E1 24.8616,E2 300.3761} C_DIS
LIN {X -64.5913,Y 40.2931,Z 82,A 141.8283,B 24.8939,C -2.3777,E1 24.865,E2 302.7041} C_DIS
LIN {X -62.8035,Y 43.0286,Z 82,A 139.2548,B 24.8936,C -2.3817,E1 24.869,E2 305.2808} C_DIS
LIN {X -59.9615,Y 46.9075,Z 82,A 135.6501,B 24.8927,C -2.3917,E1 24.875,E2 308.879} C_DIS
LIN {X -57.7965,Y 49.5497,Z 82,A 133.0908,B 24.892,C -2.3986,E1 24.8796,E2 311.4336} C_DIS
LIN {X -55.0325,Y 52.6026,Z 82,A 129.5255,B 24.8924,C -2.395,E1 24.8864,E2 315.0231} C_DIS
LIN {X -51.8034,Y 55.7869,Z 82,A 126.5102,B 24.8908,C -2.4126,E1 24.8925,E2 318.009} C_DIS
LIN {X -49.0785,Y 58.198,Z 82,A 123.6153,B 24.8906,C -2.4149,E1 24.8986,E2 320.9097} C_DIS
LIN {X -45.964,Y 60.6874,Z 82,A 120.8345,B 24.8895,C -2.4266,E1 24.9047,E2 323.6728} C_DIS
LIN {X -43.7567,Y 62.2981,Z 82,A 118.7603,B 24.8892,C -2.4303,E1 24.9094,E2 325.7454} C_DIS
LIN {X -41.1813,Y 64.0286,Z 82,A 116.4416,B 24.8887,C -2.4352,E1 24.9148,E2 328.0601} C_DIS
LIN {X -38.9491,Y 65.4109,Z 82,A 114.4534,B 24.8884,C -2.4384,E1 24.9195,E2 330.0466} C_DIS
LIN {X -36.3212,Y 66.9054,Z 82,A 112.2578,B 24.8879,C -2.4443,E1 24.9249,E2 332.2344} C_DIS
LIN {X -34.2684,Y 67.981,Z 82,A 110.4154,B 24.8879,C -2.4447,E1 24.9295,E2 334.081} C_DIS
LIN {X -31.5364,Y 69.29,Z 82,A 108.0973,B 24.8876,C -2.4472,E1 24.9353,E2 336.3989} C_DIS
LIN {X -27.1467,Y 71.1242,Z 82,A 104.5079,B 24.8872,C -2.4519,E1 24.9446,E2 339.9851} C_DIS
LIN {X -24.6322,Y 72.0342,Z 82,A 102.2196,B 24.8876,C -2.4474,E1 24.9507,E2 342.2886} C_DIS
LIN {X -20.3646,Y 73.3553,Z 82,A 99.3343,B 24.8861,C -2.4632,E1 24.9583,E2 345.1411} C_DIS
LIN {X -18.0173,Y 73.9658,Z 82,A 97.408,B 24.8861,C -2.4624,E1 24.9635,E2 347.072} C_DIS
LIN {X -14.9787,Y 74.6412,Z 82,A 94.7657,B 24.8867,C -2.4567,E1 24.9708,E2 349.7311} C_DIS
LIN {X -11.4059,Y 75.2696,Z 82,A 92.2099,B 24.8861,C -2.4632,E1 24.9778,E2 352.274} C_DIS
LIN {X -8.6608,Y 75.6346,Z 82,A 90.0277,B 24.8863,C -2.4618,E1 24.9839,E2 354.4609} C_DIS
LIN {X -5.3754,Y 75.9389,Z 82,A 87.6672,B 24.8858,C -2.4662,E1 24.9904,E2 356.8122} C_DIS
LIN {X -2.2406,Y 76.0957,Z 82,A 85.2457,B 24.8859,C -2.4654,E1 24.9972,E2 359.236} C_DIS
LIN {X 0.785,Y 76.1252,Z 82,A 82.9992,B 24.8859,C -2.4666,E1 25.0034,E2 361.4795} C_DIS
LIN {X 3.9006,Y 76.0292,Z 82,A 80.8215,B 24.8854,C -2.4712,E1 25.0095,E2 363.6455} C_DIS
LIN {X 5.9613,Y 75.8949,Z 82,A 79.1166,B 24.8858,C -2.4672,E1 25.0142,E2 365.3593} C_DIS
LIN {X 8.9002,Y 75.6065,Z 82,A 76.9406,B 24.8857,C -2.4681,E1 25.0203,E2 367.5316} C_DIS
LIN {X 12.0133,Y 75.1757,Z 82,A 74.6084,B 24.8857,C -2.4683,E1 25.0267,E2 369.8611} C_DIS
LIN {X 14.604,Y 74.715,Z 82,A 72.4547,B 24.8862,C -2.4629,E1 25.0327,E2 372.0253} C_DIS
LIN {X 17.6669,Y 74.0513,Z 82,A 70.0932,B 24.8862,C -2.4616,E1 25.0391,E2 374.3867} C_DIS
LIN {X 21.2159,Y 73.1131,Z 82,A 67.3566,B 24.8864,C -2.4605,E1 25.0464,E2 377.1214} C_DIS
LIN {X 25.9446,Y 71.5714,Z 82,A 63.707,B 24.8864,C -2.46,E1 25.0561,E2 380.7651} C_DIS
LIN {X 27.8209,Y 70.8629,Z 82,A 61.874,B 24.8874,C -2.4496,E1 25.0609,E2 382.6188} C_DIS
LIN {X 31.348,Y 69.3748,Z 82,A 59.2406,B 24.887,C -2.4533,E1 25.0676,E2 385.237} C_DIS
LIN {X 34.0422,Y 68.0937,Z 82,A 57.2872,B 24.8865,C -2.4587,E1 25.0725,E2 387.1723} C_DIS
LIN {X 37.5551,Y 66.222,Z 82,A 53.3617,B 24.8893,C -2.4286,E1 25.0822,E2 391.1577} C_DIS
LIN {X 40.5485,Y 64.4317,Z 82,A 51.5593,B 24.8875,C -2.4478,E1 25.0864,E2 392.9091} C_DIS
LIN {X 43.2075,Y 62.6798,Z 82,A 49.0319,B 24.8882,C -2.4402,E1 25.0923,E2 395.4459} C_DIS
LIN {X 45.8081,Y 60.8045,Z 82,A 46.6072,B 24.8887,C -2.4357,E1 25.0977,E2 397.8726} C_DIS
LIN {X 48.338,Y 58.8147,Z 82,A 44.1528,B 24.8892,C -2.4303,E1 25.1031,E2 400.3305} C_DIS
LIN {X 51.2875,Y 56.2602,Z 82,A 41.3115,B 24.8894,C -2.4273,E1 25.109,E2 403.1675} C_DIS
LIN {X 53.6936,Y 53.9688,Z 82,A 38.8551,B 24.8898,C -2.4234,E1 25.1139,E2 405.623} C_DIS
LIN {X 56.4711,Y 51.056,Z 82,A 35.7684,B 24.8905,C -2.4151,E1 25.1198,E2 408.7158} C_DIS
LIN {X 58.4795,Y 48.7413,Z 82,A 33.6377,B 24.8905,C -2.415,E1 25.1236,E2 410.8372} C_DIS
LIN {X 60.9698,Y 45.5881,Z 82,A 30.0376,B 24.8927,C -2.391,E1 25.1298,E2 414.4771} C_DIS
LIN {X 63.343,Y 42.2301,Z 82,A 27.3804,B 24.8923,C -2.396,E1 25.134,E2 417.1093} C_DIS
LIN {X 65.1981,Y 39.3044,Z 82,A 24.9163,B 24.8925,C -2.3934,E1 25.1376,E2 419.5669} C_DIS
LIN {X 66.6427,Y 36.8027,Z 82,A 22.8832,B 24.8926,C -2.3918,E1 25.1404,E2 421.5934} C_DIS
LIN {X 67.9044,Y 34.4182,Z 82,A 20.6736,B 24.8936,C -2.3809,E1 25.1433,E2 423.8169} C_DIS
LIN {X 69.0145,Y 32.1334,Z 82,A 18.3993,B 24.8951,C -2.3649,E1 25.146,E2 426.1169} C_DIS
LIN {X 70.7667,Y 28.0661,Z 82,A 15.4582,B 24.8949,C -2.367,E1 25.1491,E2 429.0368} C_DIS
LIN {X 71.8655,Y 25.1182,Z 82,A 13.2078,B 24.8952,C -2.3636,E1 25.1513,E2 431.2827} C_DIS
LIN {X 72.7828,Y 22.3221,Z 82,A 10.8003,B 24.8963,C -2.3512,E1 25.1533,E2 433.7057} C_DIS
LIN {X 73.6595,Y 19.2334,Z 82,A 8.829,B 24.8957,C -2.3573,E1 25.1548,E2 435.6513} C_DIS
LIN {X 74.3247,Y 16.4762,Z 82,A 6.3709,B 24.8972,C -2.341,E1 25.1563,E2 438.1336} C_DIS
LIN {X 74.9946,Y 13.0966,Z 82,A 3.7878,B 24.8978,C -2.3333,E1 25.1577,E2 440.7198} C_DIS
LIN {X 75.4727,Y 9.9737,Z 82,A 1.1791,B 24.8991,C -2.319,E1 25.1587,E2 443.347} C_DIS
LIN {X 75.8876,Y 6.0525,Z 82,A -1.3986,B 24.8989,C -2.3214,E1 25.1594,E2 445.9037} C_DIS
LIN {X 76.0663,Y 3.085,Z 82,A -3.5635,B 24.8993,C -2.3165,E1 25.1597,E2 448.0674} C_DIS
LIN {X 76.1285,Y 0.2682,Z 82,A -5.8556,B 24.9004,C -2.3045,E1 25.1597,E2 450.374} C_DIS
LIN {X 76.0728,Y -2.9326,Z 82,A -8.2489,B 24.901,C -2.2973,E1 25.1596,E2 452.7701} C_DIS
LIN {X 75.9009,Y -5.8855,Z 82,A -10.3757,B 24.9013,C -2.2932,E1 25.1592,E2 454.894} C_DIS
LIN {X 75.6397,Y -8.617,Z 82,A -12.2727,B 24.9015,C -2.2917,E1 25.1587,E2 456.7833} C_DIS
LIN {X 75.2823,Y -11.3238,Z 82,A -14.545,B 24.9026,C -2.2786,E1 25.1578,E2 459.0731} C_DIS
LIN {X 74.6728,Y -14.8229,Z 82,A -17.2505,B 24.9034,C -2.2692,E1 25.1564,E2 461.7852} C_DIS
LIN {X 74.073,Y -17.5771,Z 82,A -19.3063,B 24.9038,C -2.2644,E1 25.1551,E2 463.8401} C_DIS
LIN {X 73.3717,Y -20.3059,Z 82,A -21.4496,B 24.9044,C -2.2571,E1 25.1536,E2 465.9885} C_DIS
LIN {X 72.5994,Y -22.9137,Z 82,A -23.2282,B 24.9043,C -2.2589,E1 25.1521,E2 467.7528} C_DIS
LIN {X 71.6825,Y -25.6395,Z 82,A -25.369,B 24.9048,C -2.2529,E1 25.1502,E2 469.8957} C_DIS
LIN {X 70.3947,Y -28.9869,Z 82,A -28.137,B 24.9057,C -2.2426,E1 25.1474,E2 472.6726} C_DIS
LIN {X 69.2061,Y -31.7216,Z 82,A -30.4753,B 24.9065,C -2.233,E1 25.1447,E2 475.0208} C_DIS
LIN {X 67.9283,Y -34.3716,Z 82,A -32.3676,B 24.9062,C -2.2362,E1 25.1424,E2 476.8955} C_DIS
LIN {X 66.7538,Y -36.6,Z 82,A -34.4996,B 24.9073,C -2.2235,E1 25.1395,E2 479.0461} C_DIS
LIN {X 65.517,Y -38.7696,Z 82,A -36.6244,B 24.9083,C -2.2108,E1 25.1365,E2 481.1901} C_DIS
LIN {X 62.9771,Y -42.7722,Z 82,A -40.41,B 24.9097,C -2.1944,E1 25.1307,E2 484.9955} C_DIS
LIN {X 59.6418,Y -47.3121,Z 82,A -44.2284,B 24.9096,C -2.1956,E1 25.1243,E2 488.7929} C_DIS
LIN {X 57.6145,Y -49.7625,Z 82,A -46.6947,B 24.9103,C -2.1872,E1 25.1198,E2 491.2677} C_DIS
LIN {X 54.97,Y -52.668,Z 82,A -49.5045,B 24.9105,C -2.1843,E1 25.1145,E2 494.0722} C_DIS
LIN {X 52.7765,Y -54.8653,Z 82,A -51.8549,B 24.911,C -2.1783,E1 25.1098,E2 496.4269} C_DIS
LIN {X 50.399,Y -57.0586,Z 82,A -54.3454,B 24.9116,C -2.171,E1 25.1046,E2 498.9246} C_DIS
LIN {X 47.4528,Y -59.5306,Z 82,A -57.4936,B 24.9127,C -2.1573,E1 25.0978,E2 502.0933} C_DIS
LIN {X 44.2286,Y -61.9628,Z 82,A -60.3539,B 24.9127,C -2.1562,E1 25.0914,E2 504.9461} C_DIS
LIN {X 40.2314,Y -64.6298,Z 82,A -63.1553,B 24.9114,C -2.1729,E1 25.085,E2 507.6985} C_DIS
LIN {X 37.488,Y -66.2597,Z 82,A -66.2285,B 24.9134,C -2.149,E1 25.0774,E2 510.8189} C_DIS
LIN {X 34.673,Y -67.7742,Z 82,A -68.4677,B 24.9134,C -2.1498,E1 25.0719,E2 513.0501} C_DIS
LIN {X 32.2074,Y -68.9801,Z 82,A -70.5452,B 24.9136,C -2.1462,E1 25.0667,E2 515.1307} C_DIS
LIN {X 29.663,Y -70.1119,Z 82,A -72.7046,B 24.914,C -2.1413,E1 25.0611,E2 517.2965} C_DIS
LIN {X 26.943,Y -71.2014,Z 82,A -74.6893,B 24.9137,C -2.1445,E1 25.056,E2 519.2691} C_DIS
LIN {X 23.7034,Y -72.3449,Z 82,A -77.1506,B 24.9137,C -2.1448,E1 25.0495,E2 521.7249} C_DIS
LIN {X 20.9964,Y -73.1763,Z 82,A -79.569,B 24.9146,C -2.1342,E1 25.043,E2 524.164} C_DIS
LIN {X 18.3121,Y -73.8939,Z 82,A -81.7282,B 24.9149,C -2.1302,E1 25.0371,E2 526.3294} C_DIS
LIN {X 15.4942,Y -74.5354,Z 82,A -83.8318,B 24.9149,C -2.1302,E1 25.0314,E2 528.4303} C_DIS
LIN {X 12.6272,Y -75.0741,Z 82,A -86.0444,B 24.9151,C -2.128,E1 25.0253,E2 530.6457} C_DIS
LIN {X 9.8976,Y -75.4825,Z 82,A -88.257,B 24.9155,C -2.1229,E1 25.0192,E2 532.8685} C_DIS
LIN {X 6.4315,Y -75.8573,Z 82,A -90.8101,B 24.9155,C -2.1234,E1 25.0121,E2 535.4188} C_DIS
LIN {X 3.3236,Y -76.056,Z 82,A -92.9818,B 24.9151,C -2.1272,E1 25.0061,E2 537.5806} C_DIS
LIN {X 0.9531,Y -76.1239,Z 82,A -95.0936,B 24.9159,C -2.1178,E1 25.0001,E2 539.7146} C_DIS
LIN {X 0.9531,Y -76.1239,Z 82,A -95.0936,B 24.9159,C -2.1178,E1 25.0001,E2 539.7146} C_DIS
Enddeposition()
LIN {X 0.5084,Y -75.156,Z 82,A -95.0256,B 24.9137,C -2.1457,E1 25.0005,E2 539.5804} C_DIS
Startdeposition()
$VEL.CP = VEL_PRINT
LIN {X 2.4777,Y -75.1191,Z 82,A -92.6783,B 24.9117,C -2.1692,E1 25.0072,E2 537.1777} C_DIS
LIN {X 5.5231,Y -74.9579,Z 82,A -90.2948,B 24.9115,C -2.1718,E1 25.0138,E2 534.7891} C_DIS
LIN {X 8.5586,Y -74.6711,Z 82,A -88.0525,B 24.9116,C -2.1708,E1 25.0201,E2 532.5505} C_DIS
LIN {X 11.6462,Y -74.2521,Z 82,A -85.8136,B 24.9118,C -2.1686,E1 25.0262,E2 530.3188} C_DIS
LIN {X 14.3785,Y -73.7718,Z 82,A -83.7076,B 24.9117,C -2.1701,E1 25.032,E2 528.2117} C_DIS
LIN {X 17.0779,Y -73.194,Z 82,A -81.6063,B 24.9115,C -2.1719,E1 25.0377,E2 526.1089} C_DIS
LIN {X 19.7539,Y -72.5175,Z 82,A -79.5058,B 24.9114,C -2.174,E1 25.0434,E2 524.0067} C_DIS
LIN {X 22.0758,Y -71.8448,Z 82,A -77.5259,B 24.9109,C -2.1799,E1 25.0487,E2 522.0161} C_DIS
LIN {X 25.064,Y -70.8577,Z 82,A -75.2726,B 24.9109,C -2.1788,E1 25.0547,E2 519.77} C_DIS
LIN {X 27.3293,Y -70.0151,Z 82,A -73.3062,B 24.9105,C -2.1848,E1 25.0598,E2 517.7936} C_DIS
LIN {X 29.881,Y -68.9647,Z 82,A -71.2101,B 24.9102,C -2.1876,E1 25.0652,E2 515.6957} C_DIS
LIN {X 32.7006,Y -67.6733,Z 82,A -68.9851,B 24.9102,C -2.1873,E1 25.0708,E2 513.4772} C_DIS
LIN {X 35.1625,Y -66.4275,Z 82,A -66.7377,B 24.9096,C -2.195,E1 25.0765,E2 511.2179} C_DIS
LIN {X 37.8266,Y -64.9486,Z 82,A -64.3549,B 24.9091,C -2.2008,E1 25.0822,E2 508.8283} C_DIS
LIN {X 40.2045,Y -63.5042,Z 82,A -62.2515,B 24.9089,C -2.2043,E1 25.0872,E2 506.7235} C_DIS
LIN {X 42.4911,Y -61.9973,Z 82,A -60.2997,B 24.9089,C -2.2044,E1 25.0917,E2 504.7778} C_DIS
LIN {X 44.7113,Y -60.4155,Z 82,A -58.0808,B 24.9081,C -2.2129,E1 25.0968,E2 502.5469} C_DIS
LIN {X 47.2827,Y -58.4237,Z 82,A -55.6864,B 24.9079,C -2.2157,E1 25.102,E2 500.1547} C_DIS
LIN {X 49.6865,Y -56.3945,Z 82,A -53.2738,B 24.9074,C -2.2215,E1 25.1071,E2 497.7378} C_DIS
LIN {X 51.9312,Y -54.3345,Z 82,A -50.9778,B 24.907,C -2.2262,E1 25.1118,E2 495.4402} C_DIS
LIN {X 54.0085,Y -52.2694,Z 82,A -48.8361,B 24.9068,C -2.2289,E1 25.116,E2 493.3012} C_DIS
LIN {X 55.9977,Y -50.1322,Z 82,A -46.5705,B 24.9062,C -2.2357,E1 25.1203,E2 491.0296} C_DIS
LIN {X 58.0101,Y -47.7903,Z 82,A -44.2428,B 24.9058,C -2.241,E1 25.1245,E2 488.7001} C_DIS
LIN {X 59.8453,Y -45.4719,Z 82,A -41.9377,B 24.9052,C -2.2485,E1 25.1284,E2 486.3881} C_DIS
LIN {X 61.4589,Y -43.2664,Z 82,A -39.8565,B 24.9047,C -2.2541,E1 25.1318,E2 484.3038} C_DIS
LIN {X 62.9935,Y -41,Z 82,A -37.7812,B 24.9042,C -2.2595,E1 25.135,E2 482.2259} C_DIS
LIN {X 64.4421,Y -38.683,Z 82,A -35.7191,B 24.9038,C -2.2648,E1 25.138,E2 480.1618} C_DIS
LIN {X 65.924,Y -36.0985,Z 82,A -33.4736,B 24.9033,C -2.2706,E1 25.1411,E2 477.9143} C_DIS
LIN {X 67.4161,Y -33.2276,Z 82,A -31.2149,B 24.9032,C -2.2716,E1 25.1439,E2 475.6653} C_DIS
LIN {X 68.5903,Y -30.7308,Z 82,A -29.124,B 24.9027,C -2.2775,E1 25.1464,E2 473.5718} C_DIS
LIN {X 69.6717,Y -28.1933,Z 82,A -27.0339,B 24.9022,C -2.2835,E1 25.1486,E2 471.4791} C_DIS
LIN {X 70.6682,Y -25.5934,Z 82,A -24.9282,B 24.9017,C -2.2894,E1 25.1507,E2 469.371} C_DIS
LIN {X 71.5671,Y -22.96,Z 82,A -22.6637,B 24.9007,C -2.3003,E1 25.1527,E2 467.0936} C_DIS
LIN {X 72.4404,Y -20.0396,Z 82,A -20.2991,B 24.9,C -2.3088,E1 25.1545,E2 464.7224} C_DIS
LIN {X 73.1273,Y -17.3665,Z 82,A -18.2076,B 24.8994,C -2.3151,E1 25.1559,E2 462.6283} C_DIS
LIN {X 73.7155,Y -14.6699,Z 82,A -16.1196,B 24.8989,C -2.3212,E1 25.1571,E2 460.5379} C_DIS
LIN {X 74.251,Y -11.6534,Z 82,A -13.8746,B 24.8985,C -2.3259,E1 25.1581,E2 458.2951} C_DIS
LIN {X 74.6703,Y -8.5647,Z 82,A -11.6553,B 24.8982,C -2.3287,E1 25.1589,E2 456.0822} C_DIS
LIN {X 74.9344,Y -5.818,Z 82,A -9.5679,B 24.8977,C -2.3349,E1 25.1594,E2 453.9925} C_DIS
LIN {X 75.0828,Y -3.4049,Z 82,A -7.6019,B 24.8969,C -2.3445,E1 25.1597,E2 452.0154} C_DIS
LIN {X 75.1587,Y -0.4421,Z 82,A -5.4338,B 24.8965,C -2.349,E1 25.1597,E2 449.8498} C_DIS
LIN {X 75.119,Y 2.4807,Z 82,A -3.1259,B 24.8956,C -2.3585,E1 25.1597,E2 447.5333} C_DIS
LIN {X 74.958,Y 5.5218,Z 82,A -0.7605,B 24.8949,C -2.3671,E1 25.1592,E2 445.1614} C_DIS
LIN {X 74.6718,Y 8.5525,Z 82,A 1.4673,B 24.8945,C -2.3716,E1 25.1586,E2 442.9362} C_DIS
LIN {X 74.2503,Y 11.6582,Z 82,A 3.7011,B 24.8942,C -2.3744,E1 25.1577,E2 440.7091} C_DIS
LIN {X 73.7726,Y 14.3738,Z 82,A 5.7898,B 24.8937,C -2.3805,E1 25.1566,E2 438.6182} C_DIS
LIN {X 73.1959,Y 17.0697,Z 82,A 7.8788,B 24.8931,C -2.3865,E1 25.1554,E2 436.527} C_DIS
LIN {X 72.5149,Y 19.7636,Z 82,A 9.9845,B 24.8926,C -2.3926,E1 25.1539,E2 434.4191} C_DIS
LIN {X 71.8383,Y 22.0968,Z 82,A 11.9537,B 24.8918,C -2.4016,E1 25.1523,E2 432.4398} C_DIS
LIN {X 70.8644,Y 25.0449,Z 82,A 14.1727,B 24.8915,C -2.4042,E1 25.1503,E2 430.2273} C_DIS
LIN {X 70.0212,Y 27.3139,Z 82,A 16.1249,B 24.8908,C -2.4127,E1 25.1483,E2 428.2657} C_DIS
LIN {X 68.9982,Y 29.8044,Z 82,A 18.2205,B 24.8901,C -2.4198,E1 25.1461,E2 426.1649} C_DIS
LIN {X 67.671,Y 32.7054,Z 82,A 20.4618,B 24.8901,C -2.421,E1 25.1434,E2 423.933} C_DIS
LIN {X 66.4257,Y 35.1658,Z 82,A 22.712,B 24.8891,C -2.4311,E1 25.1405,E2 421.6707} C_DIS
LIN {X 64.9381,Y 37.8448,Z 82,A 25.0913,B 24.8884,C -2.4386,E1 25.1372,E2 419.2861} C_DIS
LIN {X 63.5037,Y 40.2054,Z 82,A 27.0759,B 24.8882,C -2.4405,E1 25.1343,E2 417.3071} C_DIS
LIN {X 61.9823,Y 42.5134,Z 82,A 29.1581,B 24.8878,C -2.445,E1 25.131,E2 415.2244} C_DIS
LIN {X 60.4081,Y 44.7214,Z 82,A 31.3547,B 24.887,C -2.4539,E1 25.1274,E2 413.0174} C_DIS
LIN {X 58.4346,Y 47.2693,Z 82,A 33.7337,B 24.8867,C -2.4575,E1 25.1233,E2 410.6411} C_DIS
LIN {X 56.4031,Y 49.6767,Z 82,A 36.1416,B 24.8861,C -2.4631,E1 25.1189,E2 408.2308} C_DIS
LIN {X 54.3306,Y 51.9352,Z 82,A 38.4518,B 24.8857,C -2.4674,E1 25.1145,E2 405.9204} C_DIS
LIN {X 52.2637,Y 54.014,Z 82,A 40.5969,B 24.8855,C -2.4695,E1 25.1102,E2 403.7794} C_DIS
LIN {X 50.1368,Y 55.9936,Z 82,A 42.8558,B 24.885,C -2.4752,E1 25.1056,E2 401.5161} C_DIS
LIN {X 47.7925,Y 58.0083,Z 82,A 45.1894,B 24.8847,C -2.479,E1 25.1006,E2 399.1826} C_DIS
LIN {X 45.5142,Y 59.8134,Z 82,A 47.4787,B 24.8841,C -2.4851,E1 25.0955,E2 396.8873} C_DIS
LIN {X 43.0485,Y 61.6104,Z 82,A 49.7231,B 24.8839,C -2.4867,E1 25.0904,E2 394.6469} C_DIS
LIN {X 40.4583,Y 63.3414,Z 82,A 52.0966,B 24.8836,C -2.4904,E1 25.0849,E2 392.2725} C_DIS
LIN {X 37.8731,Y 64.9214,Z 82,A 54.4574,B 24.8831,C -2.4952,E1 25.0792,E2 389.9077} C_DIS
LIN {X 35.4872,Y 66.2555,Z 82,A 56.526,B 24.8829,C -2.4976,E1 25.0741,E2 387.8394} C_DIS
LIN {X 33.2305,Y 67.4147,Z 82,A 58.2563,B 24.8832,C -2.4943,E1 25.0698,E2 386.1216} C_DIS
LIN {X 30.725,Y 68.5929,Z 82,A 60.3594,B 24.883,C -2.4965,E1 25.0645,E2 384.0186} C_DIS
LIN {X 28.1676,Y 69.6822,Z 82,A 62.4715,B 24.8828,C -2.4985,E1 25.0591,E2 381.9066} C_DIS
LIN {X 25.6041,Y 70.6643,Z 82,A 64.5627,B 24.8826,C -2.5004,E1 25.0536,E2 379.8154} C_DIS
LIN {X 23.0091,Y 71.5512,Z 82,A 66.7719,B 24.8822,C -2.5054,E1 25.0477,E2 377.5986} C_DIS
LIN {X 20.1183,Y 72.4181,Z 82,A 69.1437,B 24.8818,C -2.5089,E1 25.0413,E2 375.2224} C_DIS
LIN {X 17.3674,Y 73.1271,Z 82,A 71.3301,B 24.8817,C -2.5107,E1 25.0354,E2 373.0349} C_DIS
LIN {X 14.6584,Y 73.7179,Z 82,A 73.4373,B 24.8817,C -2.5115,E1 25.0297,E2 370.9285} C_DIS
LIN {X 11.6556,Y 74.2506,Z 82,A 75.6786,B 24.8817,C -2.51,E1 25.0235,E2 368.693} C_DIS
LIN {X 8.5818,Y 74.6683,Z 82,A 77.909,B 24.882,C -2.5069,E1 25.0173,E2 366.4719} C_DIS
LIN {X 5.8349,Y 74.933,Z 82,A 80.0075,B 24.882,C -2.5069,E1 25.0115,E2 364.3745} C_DIS
LIN {X 3.3984,Y 75.083,Z 82,A 82.0063,B 24.8817,C -2.5106,E1 25.0059,E2 362.3677} C_DIS
LIN {X 0.639,Y 75.1572,Z 82,A 84.1137,B 24.8817,C -2.5103,E1 25,E2 360.2611} C_DIS
LIN {X -2.4624,Y 75.1195,Z 82,A 86.4968,B 24.8817,C -2.5103,E1 24.9934,E2 357.8781} C_DIS
LIN {X -5.5294,Y 74.9575,Z 82,A 88.9052,B 24.8817,C -2.511,E1 24.9867,E2 355.4669} C_DIS
LIN {X -8.2794,Y 74.7037,Z 82,A 90.9,B 24.882,C -2.507,E1 24.9811,E2 353.4804} C_DIS
LIN {X -11.0181,Y 74.3491,Z 82,A 93.1199,B 24.8819,C -2.5087,E1 24.975,E2 351.2549} C_DIS
LIN {X -13.9922,Y 73.8461,Z 82,A 95.3662,B 24.8822,C -2.5056,E1 24.9688,E2 349.0136} C_DIS
LIN {X -17.0837,Y 73.1926,Z 82,A 97.6191,B 24.8827,C -2.4995,E1 24.9627,E2 346.7724} C_DIS
LIN {X -19.767,Y 72.514,Z 82,A 99.7189,B 24.883,C -2.4971,E1 24.957,E2 344.6751} C_DIS
LIN {X -22.3036,Y 71.7742,Z 82,A 101.8068,B 24.883,C -2.4968,E1 24.9515,E2 342.5845} C_DIS
LIN {X -25.0515,Y 70.8621,Z 82,A 103.9649,B 24.8834,C -2.4929,E1 24.9458,E2 340.4317} C_DIS
LIN {X -27.3055,Y 70.0245,Z 82,A 105.9426,B 24.8832,C -2.4941,E1 24.9406,E2 338.4468} C_DIS
LIN {X -29.8397,Y 68.9828,Z 82,A 108.045,B 24.8835,C -2.4915,E1 24.9352,E2 336.3458} C_DIS
LIN {X -32.6252,Y 67.7096,Z 82,A 110.3615,B 24.8839,C -2.4875,E1 24.9293,E2 334.033} C_DIS
LIN {X -35.17,Y 66.4235,Z 82,A 112.582,B 24.8841,C -2.4851,E1 24.9238,E2 331.8121} C_DIS
LIN {X -37.8567,Y 64.9312,Z 82,A 114.9928,B 24.8843,C -2.4827,E1 24.918,E2 329.4} C_DIS
LIN {X -40.457,Y 63.3422,Z 82,A 117.2439,B 24.8849,C -2.4767,E1 24.9127,E2 327.1563} C_DIS
LIN {X -43.0348,Y 61.6199,Z 82,A 119.4854,B 24.8856,C -2.469,E1 24.9075,E2 324.9254} C_DIS
LIN {X -44.9935,Y 60.2047,Z 82,A 121.4451,B 24.8856,C -2.4682,E1 24.9031,E2 322.9608} C_DIS
LIN {X -47.3064,Y 58.4046,Z 82,A 123.7351,B 24.886,C -2.4648,E1 24.8981,E2 320.6704} C_DIS
LIN {X -49.6769,Y 56.4029,Z 82,A 126.1464,B 24.8864,C -2.4606,E1 24.893,E2 318.2596} C_DIS
LIN {X -51.919,Y 54.3462,Z 82,A 128.4694,B 24.8868,C -2.4554,E1 24.8883,E2 315.9396} C_DIS
LIN {X -53.9927,Y 52.2858,Z 82,A 130.6297,B 24.8875,C -2.4484,E1 24.884,E2 313.7868} C_DIS
LIN {X -55.9042,Y 50.2366,Z 82,A 132.7983,B 24.8879,C -2.4439,E1 24.88,E2 311.6194} C_DIS
LIN {X -57.8897,Y 47.9351,Z 82,A 135.1833,B 24.8883,C -2.4396,E1 24.8757,E2 309.2337} C_DIS
LIN {X -59.8016,Y 45.5296,Z 82,A 137.5791,B 24.8888,C -2.4347,E1 24.8716,E2 306.8382} C_DIS
LIN {X -61.4271,Y 43.3113,Z 82,A 139.6998,B 24.8892,C -2.4296,E1 24.8681,E2 304.7193} C_DIS
LIN {X -63.001,Y 40.9886,Z 82,A 141.8449,B 24.8897,C -2.4238,E1 24.8648,E2 302.5772} C_DIS
LIN {X -64.4632,Y 38.6482,Z 82,A 143.9609,B 24.8903,C -2.4182,E1 24.8617,E2 300.4638} C_DIS
LIN {X -65.9759,Y 36.0028,Z 82,A 146.2264,B 24.891,C -2.4102,E1 24.8587,E2 298.2055} C_DIS
LIN {X -67.4166,Y 33.2266,Z 82,A 148.4807,B 24.8919,C -2.4001,E1 24.8558,E2 295.9632} C_DIS
LIN {X -68.5921,Y 30.7267,Z 82,A 150.6152,B 24.8924,C -2.3946,E1 24.8533,E2 293.8303} C_DIS
LIN {X -69.6825,Y 28.1667,Z 82,A 152.7377,B 24.893,C -2.3882,E1 24.8511,E2 291.7113} C_DIS
LIN {X -70.6674,Y 25.5956,Z 82,A 154.8496,B 24.8935,C -2.3821,E1 24.849,E2 289.6019} C_DIS
LIN {X -71.5573,Y 22.9903,Z 82,A 157.116,B 24.8937,C -2.3796,E1 24.847,E2 287.3286} C_DIS
LIN {X -72.4377,Y 20.0493,Z 82,A 159.5362,B 24.8942,C -2.3742,E1 24.8451,E2 284.9073} C_DIS
LIN {X -73.1199,Y 17.3966,Z 82,A 161.6342,B 24.8948,C -2.3679,E1 24.8437,E2 282.8121} C_DIS
LIN {X -73.7181,Y 14.6569,Z 82,A 163.7864,B 24.8954,C -2.3615,E1 24.8425,E2 280.6625} C_DIS
LIN {X -74.241,Y 11.7184,Z 82,A 166.013,B 24.8961,C -2.3532,E1 24.8415,E2 278.4426} C_DIS
LIN {X -74.6433,Y 8.7954,Z 82,A 168.2838,B 24.8967,C -2.3465,E1 24.8407,E2 276.174} C_DIS
LIN {X -74.9343,Y 5.8192,Z 82,A 170.4289,B 24.8976,C -2.3361,E1 24.8402,E2 274.041} C_DIS
LIN {X -75.0828,Y 3.4033,Z 82,A 172.4306,B 24.8978,C -2.3339,E1 24.8399,E2 272.0325} C_DIS
LIN {X -75.1588,Y 0.4254,Z 82,A 174.6342,B 24.8986,C -2.3251,E1 24.8398,E2 269.8366} C_DIS
LIN {X -75.1191,Y -2.4768,Z 82,A 176.9611,B 24.8989,C -2.3208,E1 24.8399,E2 267.506} C_DIS
LIN {X -74.9579,Y -5.5235,Z 82,A 179.365,B 24.8994,C -2.3153,E1 24.8404,E2 265.1009} C_DIS
LIN {X -74.6688,Y -8.578,Z 82,A -178.364,B 24.9002,C -2.3063,E1 24.841,E2 262.8375} C_DIS
LIN {X -74.304,Y -11.3105,Z 82,A -176.2449,B 24.9007,C -2.3002,E1 24.8419,E2 260.7204} C_DIS
LIN {X -73.7727,Y -14.3735,Z 82,A -174.0081,B 24.9016,C -2.2897,E1 24.843,E2 258.4954} C_DIS
LIN {X -73.2879,Y -16.6711,Z 82,A -172.0229,B 24.9017,C -2.2889,E1 24.8442,E2 256.5006} C_DIS
LIN {X -72.5283,Y -19.7142,Z 82,A -169.7814,B 24.9026,C -2.2781,E1 24.8457,E2 254.2717} C_DIS
LIN {X -71.8805,Y -21.9606,Z 82,A -167.792,B 24.9026,C -2.2777,E1 24.8473,E2 252.2717} C_DIS
LIN {X -70.8749,Y -25.015,Z 82,A -165.3677,B 24.9033,C -2.2699,E1 24.8495,E2 249.8524} C_DIS
LIN {X -69.7905,Y -27.9012,Z 82,A -163.0545,B 24.904,C -2.2622,E1 24.8518,E2 247.5445} C_DIS
LIN {X -68.7211,Y -30.4399,Z 82,A -160.8204,B 24.9042,C -2.2595,E1 24.8543,E2 245.3046} C_DIS
LIN {X -67.4151,Y -33.2297,Z 82,A -158.5472,B 24.9049,C -2.2512,E1 24.8571,E2 243.0389} C_DIS
LIN {X -65.9748,Y -36.0048,Z 82,A -156.2797,B 24.9057,C -2.2419,E1 24.86,E2 240.7814} C_DIS
LIN {X -64.6112,Y -38.3979,Z 82,A -154.0139,B 24.9058,C -2.2404,E1 24.8632,E2 238.5075} C_DIS
LIN {X -63.0044,Y -40.9834,Z 82,A -151.5973,B 24.9061,C -2.2368,E1 24.8668,E2 236.0873} C_DIS
LIN {X -61.2926,Y -43.4998,Z 82,A -149.3648,B 24.9068,C -2.2289,E1 24.8704,E2 233.8626} C_DIS
LIN {X -59.6411,Y -45.7379,Z 82,A -147.2352,B 24.9072,C -2.224,E1 24.874,E2 231.7345} C_DIS
LIN {X -57.4133,Y -48.5056,Z 82,A -144.4759,B 24.9076,C -2.219,E1 24.8789,E2 228.9744} C_DIS
LIN {X -55.3918,Y -50.8009,Z 82,A -142.1541,B 24.9081,C -2.2136,E1 24.8832,E2 226.655} C_DIS
LIN {X -53.2509,Y -53.0417,Z 82,A -139.8121,B 24.9085,C -2.2081,E1 24.8878,E2 224.3163} C_DIS
LIN {X -51.2657,Y -54.9628,Z 82,A -137.6868,B 24.9089,C -2.2043,E1 24.8921,E2 222.1912} C_DIS
LIN {X -49.0246,Y -56.9711,Z 82,A -135.3071,B 24.909,C -2.202,E1 24.8971,E2 219.8076} C_DIS
LIN {X -46.7208,Y -58.8742,Z 82,A -133.1011,B 24.9095,C -2.1961,E1 24.9018,E2 217.6074} C_DIS
LIN {X -44.2585,Y -60.747,Z 82,A -130.8589,B 24.9101,C -2.1891,E1 24.9068,E2 215.3739} C_DIS
LIN {X -42.004,Y -62.3272,Z 82,A -128.7501,B 24.9104,C -2.1859,E1 24.9117,E2 213.2655} C_DIS
LIN {X -40.0807,Y -63.5815,Z 82,A -126.7983,B 24.9102,C -2.1884,E1 24.9163,E2 211.3015} C_DIS
LIN {X -37.3345,Y -65.2314,Z 82,A -124.3754,B 24.9105,C -2.1844,E1 24.9221,E2 208.8807} C_DIS
LIN {X -34.6139,Y -66.7164,Z 82,A -121.9556,B 24.9106,C -2.1828,E1 24.9281,E2 206.458} C_DIS
LIN {X -32.149,Y -67.9384,Z 82,A -119.8481,B 24.9108,C -2.1806,E1 24.9334,E2 204.3504} C_DIS
LIN {X -29.6144,Y -69.081,Z 82,A -117.7299,B 24.911,C -2.1783,E1 24.9388,E2 202.2326} C_DIS
LIN {X -27.0695,Y -70.1172,Z 82,A -115.6341,B 24.9112,C -2.1764,E1 24.9443,E2 200.1369} C_DIS
LIN {X -24.4926,Y -71.0582,Z 82,A -113.5439,B 24.9113,C -2.1746,E1 24.9498,E2 198.0469} C_DIS
LIN {X -21.6295,Y -71.9807,Z 82,A -111.2758,B 24.9115,C -2.1723,E1 24.9558,E2 195.7803} C_DIS
LIN {X -18.5356,Y -72.8385,Z 82,A -109.0031,B 24.912,C -2.1662,E1 24.9619,E2 193.5186} C_DIS
LIN {X -15.849,Y -73.4699,Z 82,A -106.8983,B 24.912,C -2.1652,E1 24.9677,E2 191.4135} C_DIS
LIN {X -13.141,Y -74.0022,Z 82,A -104.637,B 24.9118,C -2.1686,E1 24.9739,E2 189.1416} C_DIS
LIN {X -10.1294,Y -74.4753,Z 82,A -102.251,B 24.9117,C -2.1697,E1 24.9805,E2 186.7509} C_DIS
LIN {X -7.3641,Y -74.7995,Z 82,A -100.1265,B 24.9117,C -2.1696,E1 24.9864,E2 184.6256} C_DIS
LIN {X -4.6137,Y -75.0194,Z 82,A -98.1351,B 24.912,C -2.1665,E1 24.9919,E2 182.6407} C_DIS
LIN {X -1.8573,Y -75.1381,Z 82,A -96.0363,B 24.912,C -2.1667,E1 24.9978,E2 180.5412} C_DIS
LIN {X 0.5084,Y -75.156,Z 82,A -95.0254,B 24.9137,C -2.1456,E1 25.0005,E2 179.5804} C_DIS
Enddeposition()
LIN {X 0.5591,Y -84.2264,Z 83,A -94.1729,B 24.9236,C -2.0186,E1 25.002,E2 179.0292} C_DIS
Startdeposition()
$VEL.CP = VEL_PRINT
LIN {X -1.5737,Y -84.2161,Z 83,A -96.2642,B 24.9251,C -1.9986,E1 24.996,E2 181.168} C_DIS
LIN {X -4.7273,Y -84.098,Z 83,A -98.392,B 24.9251,C -1.999,E1 24.9901,E2 183.2955} C_DIS
LIN {X -7.8195,Y -83.8671,Z 83,A -100.5017,B 24.9251,C -1.999,E1 24.9842,E2 185.406} C_DIS
LIN {X -10.7459,Y -83.5425,Z 83,A -102.5604,B 24.9251,C -1.9977,E1 24.9785,E2 187.4693} C_DIS
LIN {X -13.9679,Y -83.0646,Z 83,A -104.7224,B 24.9251,C -1.9999,E1 24.9726,E2 189.628} C_DIS
LIN {X -17.0158,Y -82.4942,Z 83,A -106.8336,B 24.925,C -2.0006,E1 24.9668,E2 191.7397} C_DIS
LIN {X -19.8887,Y -81.8491,Z 83,A -108.8937,B 24.925,C -1.9999,E1 24.9612,E2 193.8043} C_DIS
LIN {X -23.0384,Y -81.0189,Z 83,A -111.0574,B 24.9248,C -2.0028,E1 24.9553,E2 195.9644} C_DIS
LIN {X -26.0048,Y -80.116,Z 83,A -113.1702,B 24.9247,C -2.0043,E1 24.9497,E2 198.0774} C_DIS
LIN {X -28.695,Y -79.1925,Z 83,A -115.1474,B 24.9247,C -2.0046,E1 24.9445,E2 200.0577} C_DIS
LIN {X -31.6832,Y -78.0449,Z 83,A -117.346,B 24.9245,C -2.0061,E1 24.9388,E2 202.2576} C_DIS
LIN {X -34.5343,Y -76.8258,Z 83,A -119.4604,B 24.9244,C -2.0082,E1 24.9334,E2 204.3719} C_DIS
LIN {X -37.4788,Y -75.4332,Z 83,A -121.6268,B 24.9241,C -2.0123,E1 24.9279,E2 206.5343} C_DIS
LIN {X -40.0924,Y -74.0772,Z 83,A -123.6906,B 24.9241,C -2.0131,E1 24.9228,E2 208.6019} C_DIS
LIN {X -42.7918,Y -72.5513,Z 83,A -125.8065,B 24.9238,C -2.0158,E1 24.9177,E2 210.7175} C_DIS
LIN {X -45.5649,Y -70.8426,Z 83,A -127.9643,B 24.9234,C -2.0208,E1 24.9126,E2 212.8703} C_DIS
LIN {X -48.0131,Y -69.2067,Z 83,A -130.0399,B 24.9234,C -2.022,E1 24.9078,E2 214.9501} C_DIS
LIN {X -50.6529,Y -67.2986,Z 83,A -132.2087,B 24.923,C -2.0271,E1 24.9029,E2 217.1144} C_DIS
LIN {X -53.0957,Y -65.3887,Z 83,A -134.3267,B 24.9227,C -2.0306,E1 24.8983,E2 219.2317} C_DIS
LIN {X -55.4665,Y -63.39,Z 83,A -136.445,B 24.9224,C -2.0344,E1 24.8938,E2 221.3493} C_DIS
LIN {X -57.7621,Y -61.3055,Z 83,A -138.5636,B 24.9221,C -2.0383,E1 24.8895,E2 223.4671} C_DIS
LIN {X -59.9795,Y -59.1379,Z 83,A -140.6828,B 24.9218,C -2.0425,E1 24.8853,E2 225.5855} C_DIS
LIN {X -62.1155,Y -56.8902,Z 83,A -142.8023,B 24.9214,C -2.0468,E1 24.8812,E2 227.704} C_DIS
LIN {X -64.1674,Y -54.5653,Z 83,A -144.9205,B 24.9211,C -2.0513,E1 24.8773,E2 229.821} C_DIS
LIN {X -66.1323,Y -52.1665,Z 83,A -147.0428,B 24.9207,C -2.0558,E1 24.8736,E2 231.9423} C_DIS
LIN {X -68.0076,Y -49.697,Z 83,A -149.1633,B 24.9204,C -2.0606,E1 24.8701,E2 234.0616} C_DIS
LIN {X -69.7907,Y -47.1602,Z 83,A -151.2845,B 24.92,C -2.0656,E1 24.8667,E2 236.1814} C_DIS
LIN {X -71.4793,Y -44.5594,Z 83,A -153.406,B 24.9196,C -2.0707,E1 24.8635,E2 238.3015} C_DIS
LIN {X -73.0709,Y -41.8983,Z 83,A -155.5278,B 24.9192,C -2.0759,E1 24.8605,E2 240.4219} C_DIS
LIN {X -74.4907,Y -39.3188,Z 83,A -157.598,B 24.9189,C -2.0794,E1 24.8578,E2 242.4946} C_DIS
LIN {X -75.8874,Y -36.5503,Z 83,A -159.7206,B 24.9185,C -2.0849,E1 24.8551,E2 244.6156} C_DIS
LIN {X -77.1813,Y -33.7324,Z 83,A -161.8432,B 24.918,C -2.0905,E1 24.8527,E2 246.7365} C_DIS
LIN {X -78.3706,Y -30.8687,Z 83,A -163.9662,B 24.9176,C -2.0962,E1 24.8505,E2 248.8577} C_DIS
LIN {X -79.4537,Y -27.9632,Z 83,A -166.089,B 24.9171,C -2.102,E1 24.8485,E2 250.9788} C_DIS
LIN {X -80.4291,Y -25.0197,Z 83,A -168.2125,B 24.9167,C -2.1078,E1 24.8467,E2 253.1004} C_DIS
LIN {X -81.3363,Y -21.8914,Z 83,A -170.3877,B 24.9161,C -2.1156,E1 24.845,E2 255.2697} C_DIS
LIN {X -82.0517,Y -19.0352,Z 83,A -172.4597,B 24.9157,C -2.1198,E1 24.8436,E2 257.3437} C_DIS
LIN {X -82.6968,Y -16.0022,Z 83,A -174.5834,B 24.9152,C -2.1259,E1 24.8425,E2 259.4654} C_DIS
LIN {X -83.2536,Y -12.7929,Z 83,A -176.7205,B 24.9145,C -2.1349,E1 24.8415,E2 261.5937} C_DIS
LIN {X -83.6499,Y -9.8753,Z 83,A -178.8315,B 24.9142,C -2.1383,E1 24.8407,E2 263.7093} C_DIS
LIN {X -83.9692,Y -6.6337,Z 83,A 178.9924,B 24.9136,C -2.1464,E1 24.8402,E2 265.8792} C_DIS
LIN {X -84.1564,Y -3.5386,Z 83,A 176.8681,B 24.9131,C -2.1526,E1 24.8399,E2 268.0013} C_DIS
LIN {X -84.2299,Y -0.4893,Z 83,A 174.7407,B 24.9127,C -2.1578,E1 24.8398,E2 270.1291} C_DIS
LIN {X -84.1887,Y 2.662,Z 83,A 172.6194,B 24.9121,C -2.1653,E1 24.8399,E2 272.2454} C_DIS
LIN {X -84.0443,Y 5.6028,Z 83,A 170.5468,B 24.9117,C -2.1698,E1 24.8402,E2 274.3197} C_DIS
LIN {X -83.7811,Y 8.6924,Z 83,A 168.4223,B 24.9112,C -2.1761,E1 24.8408,E2 276.4418} C_DIS
LIN {X -83.3824,Y 11.9252,Z 83,A 166.2463,B 24.9105,C -2.1842,E1 24.8416,E2 278.6115} C_DIS
LIN {X -82.8869,Y 14.9862,Z 83,A 164.122,B 24.91,C -2.1905,E1 24.8426,E2 280.7333} C_DIS
LIN {X -82.3125,Y 17.874,Z 83,A 162.0493,B 24.9096,C -2.195,E1 24.8437,E2 282.8075} C_DIS
LIN {X -81.5988,Y 20.8916,Z 83,A 159.9252,B 24.9091,C -2.2012,E1 24.8452,E2 284.9292} C_DIS
LIN {X -80.7746,Y 23.8809,Z 83,A 157.801,B 24.9086,C -2.2074,E1 24.8468,E2 287.0509} C_DIS
LIN {X -79.8409,Y 26.8378,Z 83,A 155.6773,B 24.9081,C -2.2136,E1 24.8486,E2 289.1722} C_DIS
LIN {X -78.7989,Y 29.7583,Z 83,A 153.5534,B 24.9076,C -2.2196,E1 24.8506,E2 291.2936} C_DIS
LIN {X -77.6502,Y 32.6385,Z 83,A 151.4298,B 24.9071,C -2.2256,E1 24.8529,E2 293.4148} C_DIS
LIN {X -76.3963,Y 35.4745,Z 83,A 149.3064,B 24.9066,C -2.2315,E1 24.8553,E2 295.5356} C_DIS
LIN {X -75.0388,Y 38.2624,Z 83,A 147.1831,B 24.9061,C -2.2374,E1 24.858,E2 297.6564} C_DIS
LIN {X -73.5033,Y 41.135,Z 83,A 145.0083,B 24.9055,C -2.2449,E1 24.8609,E2 299.8248} C_DIS
LIN {X -71.9394,Y 43.8126,Z 83,A 142.886,B 24.905,C -2.2505,E1 24.8639,E2 301.9446} C_DIS
LIN {X -70.3642,Y 46.3002,Z 83,A 140.8151,B 24.9047,C -2.2543,E1 24.867,E2 304.017} C_DIS
LIN {X -68.5215,Y 48.9861,Z 83,A 138.6412,B 24.9041,C -2.2614,E1 24.8705,E2 306.1845} C_DIS
LIN {X -66.672,Y 51.475,Z 83,A 136.5191,B 24.9036,C -2.2667,E1 24.874,E2 308.3042} C_DIS
LIN {X -64.7322,Y 53.8941,Z 83,A 134.3977,B 24.9032,C -2.2718,E1 24.8778,E2 310.4232} C_DIS
LIN {X -62.7046,Y 56.2402,Z 83,A 132.2763,B 24.9027,C -2.2768,E1 24.8817,E2 312.5423} C_DIS
LIN {X -60.7007,Y 58.3974,Z 83,A 130.2072,B 24.9025,C -2.2799,E1 24.8856,E2 314.613} C_DIS
LIN {X -58.3974,Y 60.7007,Z 83,A 128.035,B 24.9019,C -2.2864,E1 24.89,E2 316.779} C_DIS
LIN {X -56.2402,Y 62.7046,Z 83,A 125.9664,B 24.9017,C -2.2892,E1 24.8942,E2 318.8492} C_DIS
LIN {X -53.8941,Y 64.7322,Z 83,A 123.8466,B 24.9013,C -2.2936,E1 24.8987,E2 320.9668} C_DIS
LIN {X -51.475,Y 66.672,Z 83,A 121.7272,B 24.9009,C -2.2978,E1 24.9034,E2 323.0839} C_DIS
LIN {X -48.9861,Y 68.5215,Z 83,A 119.6083,B 24.9006,C -2.3018,E1 24.9081,E2 325.2007} C_DIS
LIN {X -46.3002,Y 70.3642,Z 83,A 117.4384,B 24.9001,C -2.3074,E1 24.9132,E2 327.3646} C_DIS
LIN {X -43.6789,Y 72.0207,Z 83,A 115.3202,B 24.8998,C -2.311,E1 24.9182,E2 329.4807} C_DIS
LIN {X -41.135,Y 73.5033,Z 83,A 113.254,B 24.8996,C -2.3128,E1 24.9232,E2 331.5489} C_DIS
LIN {X -38.2624,Y 75.0388,Z 83,A 111.0853,B 24.8992,C -2.3177,E1 24.9285,E2 333.7117} C_DIS
LIN {X -35.4745,Y 76.3963,Z 83,A 108.9688,B 24.8989,C -2.3208,E1 24.9339,E2 335.8263} C_DIS
LIN {X -32.7827,Y 77.5895,Z 83,A 106.9041,B 24.8989,C -2.322,E1 24.9392,E2 337.8931} C_DIS
LIN {X -29.7583,Y 78.7989,Z 83,A 104.737,B 24.8985,C -2.3263,E1 24.9448,E2 340.0545} C_DIS
LIN {X -26.8378,Y 79.8409,Z 83,A 102.6248,B 24.8982,C -2.3288,E1 24.9503,E2 342.1649} C_DIS
LIN {X -23.8809,Y 80.7746,Z 83,A 100.5073,B 24.8981,C -2.331,E1 24.956,E2 344.281} C_DIS
LIN {X -21.0431,Y 81.5599,Z 83,A 98.4447,B 24.8981,C -2.3313,E1 24.9616,E2 346.346} C_DIS
LIN {X -17.874,Y 82.3125,Z 83,A 96.2795,B 24.8977,C -2.3347,E1 24.9674,E2 348.5057} C_DIS
LIN {X -14.9862,Y 82.8869,Z 83,A 94.218,B 24.8977,C -2.3346,E1 24.9731,E2 350.5698} C_DIS
LIN {X -11.9252,Y 83.3824,Z 83,A 92.1052,B 24.8977,C -2.3359,E1 24.9789,E2 352.6813} C_DIS
LIN {X -8.6924,Y 83.7811,Z 83,A 89.9422,B 24.8974,C -2.3387,E1 24.9849,E2 354.8391} C_DIS
LIN {X -5.6028,Y 84.0443,Z 83,A 87.8307,B 24.8973,C -2.3396,E1 24.9908,E2 356.9495} C_DIS
LIN {X -2.662,Y 84.1887,Z 83,A 85.771,B 24.8973,C -2.3385,E1 24.9965,E2 359.0121} C_DIS
LIN {X 0.4386,Y 84.2297,Z 83,A 83.6606,B 24.8973,C -2.3389,E1 25.0024,E2 361.1214} C_DIS
LIN {X 3.5386,Y 84.1564,Z 83,A 81.5508,B 24.8973,C -2.3391,E1 25.0083,E2 363.2303} C_DIS
LIN {X 6.6337,Y 83.9692,Z 83,A 79.4416,B 24.8973,C -2.3391,E1 25.0142,E2 365.3387} C_DIS
LIN {X 9.8753,Y 83.6499,Z 83,A 77.2819,B 24.8973,C -2.3404,E1 25.0202,E2 367.4937} C_DIS
LIN {X 12.7929,Y 83.2536,Z 83,A 75.2248,B 24.8974,C -2.3383,E1 25.0259,E2 369.5541} C_DIS
LIN {X 16.0022,Y 82.6968,Z 83,A 73.066,B 24.8974,C -2.3392,E1 25.0318,E2 371.7084} C_DIS
LIN {X 19.0352,Y 82.0517,Z 83,A 70.9588,B 24.8974,C -2.3382,E1 25.0375,E2 373.8151} C_DIS
LIN {X 21.8914,Y 81.3363,Z 83,A 68.9035,B 24.8977,C -2.3354,E1 25.0431,E2 375.8739} C_DIS
LIN {X 24.9555,Y 80.449,Z 83,A 66.7693,B 24.8977,C -2.3349,E1 25.0488,E2 378.0055} C_DIS
LIN {X 27.8155,Y 79.5055,Z 83,A 64.692,B 24.8979,C -2.3323,E1 25.0543,E2 380.085} C_DIS
LIN {X 30.8687,Y 78.3706,Z 83,A 62.5359,B 24.8979,C -2.332,E1 25.0599,E2 382.237} C_DIS
LIN {X 33.5889,Y 77.2438,Z 83,A 60.4827,B 24.8983,C -2.3283,E1 25.0652,E2 384.2941} C_DIS
LIN {X 36.5503,Y 75.8874,Z 83,A 58.3278,B 24.8983,C -2.3276,E1 25.0707,E2 386.4451} C_DIS
LIN {X 39.3188,Y 74.4907,Z 83,A 56.2244,B 24.8986,C -2.3251,E1 25.0759,E2 388.5487} C_DIS
LIN {X 42.0339,Y 72.993,Z 83,A 54.1214,B 24.8988,C -2.3224,E1 25.081,E2 390.652} C_DIS
LIN {X 44.6921,Y 71.3964,Z 83,A 52.0189,B 24.8991,C -2.3194,E1 25.086,E2 392.7548} C_DIS
LIN {X 47.2423,Y 69.7351,Z 83,A 49.9367,B 24.8994,C -2.3158,E1 25.0909,E2 394.8388} C_DIS
LIN {X 49.697,Y 68.0076,Z 83,A 47.8667,B 24.8998,C -2.3114,E1 25.0956,E2 396.9119} C_DIS
LIN {X 52.1665,Y 66.1323,Z 83,A 45.7657,B 24.9001,C -2.3079,E1 25.1002,E2 399.0135} C_DIS
LIN {X 54.6844,Y 64.0659,Z 83,A 43.6139,B 24.9003,C -2.3058,E1 25.1048,E2 401.1621} C_DIS
LIN {X 56.8632,Y 62.1403,Z 83,A 41.5757,B 24.9008,C -2.2999,E1 25.1091,E2 403.206} C_DIS
LIN {X 59.1379,Y 59.9795,Z 83,A 39.4652,B 24.9011,C -2.2962,E1 25.1133,E2 405.3163} C_DIS
LIN {X 61.3055,Y 57.7621,Z 83,A 37.366,B 24.9014,C -2.292,E1 25.1174,E2 407.4165} C_DIS
LIN {X 63.493,Y 55.3486,Z 83,A 35.2158,B 24.9017,C -2.2892,E1 25.1214,E2 409.5638} C_DIS
LIN {X 65.3887,Y 53.0957,Z 83,A 33.1684,B 24.9022,C -2.2831,E1 25.125,E2 411.6163} C_DIS
LIN {X 67.2986,Y 50.6529,Z 83,A 31.0704,B 24.9026,C -2.2783,E1 25.1286,E2 413.7154} C_DIS
LIN {X 69.1174,Y 48.1415,Z 83,A 28.9732,B 24.903,C -2.2735,E1 25.132,E2 415.8139} C_DIS
LIN {X 70.8426,Y 45.5649,Z 83,A 26.9016,B 24.9034,C -2.2694,E1 25.1352,E2 417.8849} C_DIS
LIN {X 72.4717,Y 42.9265,Z 83,A 24.7778,B 24.9039,C -2.2633,E1 25.1382,E2 420.0121} C_DIS
LIN {X 74.0772,Y 40.0924,Z 83,A 22.6297,B 24.9042,C -2.2596,E1 25.1412,E2 422.1578} C_DIS
LIN {X 75.4332,Y 37.4788,Z 83,A 20.5843,B 24.9048,C -2.2527,E1 25.1438,E2 424.2086} C_DIS
LIN {X 76.7456,Y 34.7123,Z 83,A 18.4993,B 24.9053,C -2.2468,E1 25.1462,E2 426.2963} C_DIS
LIN {X 78.0449,Y 31.6832,Z 83,A 16.3409,B 24.9056,C -2.2431,E1 25.1485,E2 428.4516} C_DIS
LIN {X 79.1046,Y 28.9361,Z 83,A 14.296,B 24.9062,C -2.2359,E1 25.1506,E2 430.5021} C_DIS
LIN {X 80.116,Y 26.0048,Z 83,A 12.2004,B 24.9067,C -2.2301,E1 25.1524,E2 432.5995} C_DIS
LIN {X 81.0189,Y 23.0384,Z 83,A 10.1049,B 24.9072,C -2.2242,E1 25.1541,E2 434.697} C_DIS
LIN {X 81.8491,Y 19.8887,Z 83,A 7.9588,B 24.9076,C -2.2198,E1 25.1556,E2 436.8411} C_DIS
LIN {X 82.5256,Y 16.8626,Z 83,A 5.8638,B 24.9081,C -2.2138,E1 25.1568,E2 438.9381} C_DIS
LIN {X 83.0646,Y 13.9679,Z 83,A 3.8195,B 24.9087,C -2.2062,E1 25.1578,E2 440.9884} C_DIS
LIN {X 83.5425,Y 10.7459,Z 83,A 1.6859,B 24.909,C -2.202,E1 25.1586,E2 443.1193} C_DIS
LIN {X 83.8671,Y 7.8195,Z 83,A -0.3699,B 24.9097,C -2.1939,E1 25.1592,E2 445.182} C_DIS
LIN {X 84.098,Y 4.7272,Z 83,A -2.4645,B 24.9102,C -2.1877,E1 25.1596,E2 447.2788} C_DIS
LIN {X 84.2151,Y 1.6286,Z 83,A -4.5599,B 24.9107,C -2.1815,E1 25.1598,E2 449.3765} C_DIS
LIN {X 84.207,Y -2.0672,Z 83,A -7.1126,B 24.9115,C -2.1721,E1 25.1597,E2 451.9361} C_DIS
LIN {X 84.0796,Y -5.0609,Z 83,A -9.1464,B 24.912,C -2.1658,E1 25.1594,E2 453.9728} C_DIS
LIN {X 83.8267,Y -8.2562,Z 83,A -11.3152,B 24.9126,C -2.1592,E1 25.1589,E2 456.1443} C_DIS
LIN {X 83.5003,Y -11.0719,Z 83,A -13.2549,B 24.9131,C -2.1526,E1 25.1582,E2 458.088} C_DIS
LIN {X 82.9923,Y -14.4005,Z 83,A -15.5349,B 24.9137,C -2.1457,E1 25.1572,E2 460.3711} C_DIS
LIN {X 82.406,Y -17.4455,Z 83,A -17.6294,B 24.9142,C -2.1395,E1 25.156,E2 462.468} C_DIS
LIN {X 81.708,Y -20.4668,Z 83,A -19.6802,B 24.9145,C -2.1348,E1 25.1546,E2 464.518} C_DIS
LIN {X 80.8993,Y -23.4604,Z 83,A -21.8189,B 24.9151,C -2.1272,E1 25.153,E2 466.6624} C_DIS
LIN {X 79.981,Y -26.4222,Z 83,A -23.914,B 24.9156,C -2.1211,E1 25.1512,E2 468.7599} C_DIS
LIN {X 78.9543,Y -29.3481,Z 83,A -26.0089,B 24.9161,C -2.1151,E1 25.1492,E2 470.8573} C_DIS
LIN {X 77.8205,Y -32.2343,Z 83,A -28.1042,B 24.9166,C -2.1091,E1 25.147,E2 472.9551} C_DIS
LIN {X 76.5814,Y -35.0768,Z 83,A -30.1996,B 24.917,C -2.1033,E1 25.1446,E2 475.0529} C_DIS
LIN {X 75.2384,Y -37.8718,Z 83,A -32.2954,B 24.9175,C -2.0974,E1 25.1421,E2 477.1513} C_DIS
LIN {X 73.7934,Y -40.6155,Z 83,A -34.3471,B 24.9178,C -2.0932,E1 25.1393,E2 479.2022} C_DIS
LIN {X 72.2485,Y -43.3041,Z 83,A -36.4433,B 24.9183,C -2.0876,E1 25.1364,E2 481.3008} C_DIS
LIN {X 70.6128,Y -45.9228,Z 83,A -38.5313,B 24.9187,C -2.0821,E1 25.1332,E2 483.3914} C_DIS
LIN {X 68.8671,Y -48.5017,Z 83,A -40.6363,B 24.9191,C -2.0767,E1 25.1299,E2 485.4987} C_DIS
LIN {X 67.0352,Y -51.0036,Z 83,A -42.7329,B 24.9195,C -2.0714,E1 25.1264,E2 487.5978} C_DIS
LIN {X 65.1125,Y -53.4364,Z 83,A -44.8301,B 24.9199,C -2.0663,E1 25.1227,E2 489.6974} C_DIS
LIN {X 63.1015,Y -55.7968,Z 83,A -46.9277,B 24.9203,C -2.0613,E1 25.1189,E2 491.7973} C_DIS
LIN {X 61.1395,Y -57.9387,Z 83,A -48.917,B 24.9207,C -2.0559,E1 25.1151,E2 493.7905} C_DIS
LIN {X 58.8259,Y -60.2877,Z 83,A -51.1237,B 24.9211,C -2.0517,E1 25.1107,E2 495.998} C_DIS
LIN {X 56.567,Y -62.4121,Z 83,A -53.2221,B 24.9214,C -2.0471,E1 25.1064,E2 498.0986} C_DIS
LIN {X 54.2314,Y -64.4518,Z 83,A -55.321,B 24.9218,C -2.0427,E1 25.1019,E2 500.1998} C_DIS
LIN {X 51.8224,Y -66.4043,Z 83,A -57.4204,B 24.9221,C -2.0385,E1 25.0973,E2 502.3014} C_DIS
LIN {X 49.3431,Y -68.2667,Z 83,A -59.5641,B 24.9225,C -2.033,E1 25.0925,E2 504.4504} C_DIS
LIN {X 46.797,Y -70.0366,Z 83,A -61.6202,B 24.9227,C -2.0305,E1 25.0877,E2 506.5054} C_DIS
LIN {X 44.1874,Y -71.7116,Z 83,A -63.7649,B 24.9231,C -2.0254,E1 25.0827,E2 508.6554} C_DIS
LIN {X 41.518,Y -73.2895,Z 83,A -65.8659,B 24.9233,C -2.0218,E1 25.0776,E2 510.7584} C_DIS
LIN {X 38.7923,Y -74.768,Z 83,A -67.9232,B 24.9235,C -2.0199,E1 25.0725,E2 512.8144} C_DIS
LIN {X 36.014,Y -76.1451,Z 83,A -70.0693,B 24.9238,C -2.0154,E1 25.0671,E2 514.9656} C_DIS
LIN {X 33.1869,Y -77.4191,Z 83,A -72.1717,B 24.9241,C -2.0125,E1 25.0617,E2 517.0698} C_DIS
Enddeposition()
END
